Yaskawa INFORM job: DEMO_ROOF_SIDE_0625_3PAINT_10.JBI

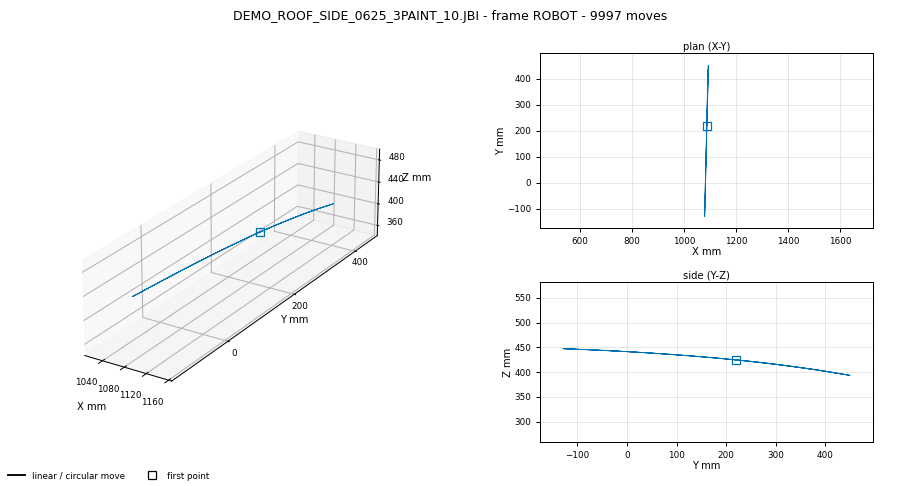
[picture p0: tool path of DEMO_ROOF_SIDE_0625_3PAINT_10.JBI in frame ROBOT, 9997 of 9997 moves have a stored position in this frame; points joined in program order, loops and branches not executed]
/JOB
//NAME DEMO_ROOF_SIDE_0625_3PAINT10
//POS
///NPOS 9997,0,0,0,0,0
///TOOL 0
///USER 0
///POSTYPE ROBOT
///RECTAN
///RCONF 1,0,0,0,0,0,0,0,0,0,0,0,0,0,0,0,0,0,0,0,0,0,0,0
C00000=1088.381,219.309,425.183,176.120,21.168,153.279
C00001=1088.386,219.557,425.158,176.123,21.170,153.279
C00002=1088.393,219.806,425.133,176.125,21.172,153.279
C00003=1088.398,220.056,425.108,176.128,21.175,153.279
C00004=1088.403,220.304,425.083,176.131,21.177,153.279
C00005=1088.409,220.553,425.058,176.134,21.180,153.280
C00006=1088.415,220.801,425.033,176.136,21.182,153.280
C00007=1088.420,221.050,425.007,176.140,21.184,153.280
C00008=1088.426,221.299,424.982,176.142,21.187,153.280
C00009=1088.432,221.547,424.957,176.145,21.189,153.280
C00010=1088.437,221.796,424.931,176.147,21.192,153.280
C00011=1088.446,222.184,424.893,176.152,21.195,153.280
C00012=1088.455,222.571,424.853,176.156,21.199,153.280
C00013=1088.463,222.958,424.814,176.160,21.203,153.280
C00014=1088.472,223.347,424.775,176.164,21.207,153.281
C00015=1088.478,223.596,424.749,176.167,21.209,153.281
C00016=1088.483,223.844,424.724,176.170,21.212,153.281
C00017=1088.490,224.092,424.698,176.173,21.214,153.281
C00018=1088.495,224.342,424.673,176.175,21.217,153.281
C00019=1088.500,224.590,424.648,176.178,21.219,153.281
C00020=1088.506,224.839,424.622,176.181,21.222,153.281
C00021=1088.511,225.087,424.597,176.184,21.224,153.281
C00022=1088.517,225.336,424.571,176.187,21.227,153.281
C00023=1088.523,225.584,424.546,176.189,21.229,153.281
C00024=1088.528,225.833,424.521,176.192,21.231,153.281
C00025=1088.534,226.082,424.496,176.195,21.233,153.281
C00026=1088.539,226.331,424.470,176.198,21.236,153.282
C00027=1088.546,226.580,424.445,176.200,21.238,153.282
C00028=1088.550,226.828,424.419,176.203,21.241,153.282
C00029=1088.557,227.077,424.394,176.205,21.243,153.282
C00030=1088.562,227.326,424.368,176.208,21.246,153.282
C00031=1088.568,227.574,424.343,176.211,21.248,153.282
C00032=1088.573,227.823,424.317,176.214,21.251,153.282
C00033=1088.579,228.071,424.292,176.217,21.253,153.282
C00034=1088.585,228.320,424.266,176.219,21.255,153.282
C00035=1088.590,228.568,424.241,176.222,21.258,153.282
C00036=1088.596,228.817,424.215,176.225,21.260,153.283
C00037=1088.601,229.066,424.189,176.228,21.263,153.283
C00038=1088.608,229.315,424.163,176.230,21.265,153.283
C00039=1088.612,229.563,424.138,176.233,21.268,153.283
C00040=1088.619,229.811,424.112,176.236,21.270,153.283
C00041=1088.624,230.060,424.086,176.239,21.273,153.283
C00042=1088.631,230.309,424.061,176.242,21.275,153.283
C00043=1088.636,230.558,424.035,176.244,21.277,153.283
C00044=1088.641,230.806,424.009,176.247,21.280,153.283
C00045=1088.646,231.055,423.983,176.250,21.282,153.283
C00046=1088.653,231.304,423.958,176.253,21.285,153.283
C00047=1088.658,231.552,423.931,176.255,21.287,153.284
C00048=1088.663,231.800,423.906,176.258,21.289,153.284
C00049=1088.669,232.049,423.880,176.261,21.292,153.284
C00050=1088.675,232.298,423.854,176.264,21.295,153.284
C00051=1088.680,232.547,423.828,176.267,21.297,153.284
C00052=1088.686,232.795,423.802,176.269,21.299,153.284
C00053=1088.692,233.043,423.777,176.272,21.302,153.284
C00054=1088.697,233.292,423.751,176.275,21.305,153.284
C00055=1088.703,233.541,423.724,176.278,21.307,153.284
C00056=1088.709,233.790,423.698,176.281,21.310,153.284
C00057=1088.714,234.039,423.672,176.283,21.312,153.285
C00058=1088.720,234.287,423.647,176.286,21.314,153.285
C00059=1088.725,234.535,423.621,176.288,21.317,153.285
C00060=1088.731,234.784,423.595,176.292,21.319,153.285
C00061=1088.737,235.032,423.568,176.295,21.322,153.285
C00062=1088.742,235.281,423.542,176.297,21.324,153.285
C00063=1088.751,235.661,423.502,176.302,21.328,153.285
C00064=1088.759,236.040,423.463,176.306,21.332,153.285
C00065=1088.768,236.419,423.422,176.310,21.336,153.286
C00066=1088.776,236.797,423.383,176.314,21.339,153.286
C00067=1088.782,237.046,423.357,176.317,21.342,153.286
C00068=1088.788,237.295,423.331,176.319,21.345,153.286
C00069=1088.793,237.544,423.305,176.323,21.347,153.286
C00070=1088.799,237.792,423.278,176.326,21.350,153.286
C00071=1088.804,238.041,423.252,176.328,21.352,153.286
C00072=1088.810,238.289,423.225,176.331,21.355,153.286
C00073=1088.816,238.538,423.199,176.334,21.357,153.286
C00074=1088.821,238.786,423.174,176.337,21.359,153.286
C00075=1088.827,239.034,423.147,176.340,21.362,153.287
C00076=1088.833,239.283,423.121,176.342,21.364,153.287
C00077=1088.838,239.531,423.094,176.345,21.367,153.287
C00078=1088.844,239.780,423.069,176.348,21.369,153.287
C00079=1088.850,240.029,423.042,176.350,21.372,153.287
C00080=1088.855,240.277,423.015,176.354,21.375,153.287
C00081=1088.861,240.526,422.989,176.357,21.377,153.287
C00082=1088.867,240.774,422.963,176.359,21.379,153.287
C00083=1088.873,241.023,422.936,176.362,21.382,153.287
C00084=1088.878,241.272,422.910,176.364,21.384,153.288
C00085=1088.884,241.520,422.883,176.368,21.387,153.288
C00086=1088.890,241.769,422.857,176.371,21.389,153.288
C00087=1088.895,242.017,422.830,176.373,21.392,153.288
C00088=1088.901,242.266,422.804,176.376,21.394,153.288
C00089=1088.906,242.515,422.777,176.379,21.397,153.288
C00090=1088.912,242.763,422.750,176.382,21.399,153.288
C00091=1088.917,243.011,422.724,176.385,21.402,153.288
C00092=1088.923,243.260,422.698,176.388,21.405,153.288
C00093=1088.929,243.509,422.671,176.390,21.407,153.288
C00094=1088.934,243.757,422.644,176.393,21.410,153.289
C00095=1088.940,244.005,422.618,176.396,21.412,153.289
C00096=1088.945,244.254,422.591,176.399,21.414,153.289
C00097=1088.951,244.502,422.564,176.402,21.417,153.289
C00098=1088.956,244.751,422.538,176.405,21.420,153.289
C00099=1088.962,245.000,422.511,176.407,21.422,153.289
C00100=1088.969,245.249,422.484,176.410,21.425,153.289
C00101=1088.974,245.497,422.457,176.413,21.428,153.289
C00102=1088.979,245.746,422.430,176.416,21.430,153.289
C00103=1088.985,245.994,422.404,176.419,21.432,153.290
C00104=1088.991,246.242,422.377,176.422,21.435,153.290
C00105=1088.996,246.491,422.350,176.424,21.437,153.290
C00106=1089.002,246.740,422.323,176.427,21.440,153.290
C00107=1089.008,246.988,422.297,176.430,21.443,153.290
C00108=1089.013,247.237,422.269,176.433,21.445,153.290
C00109=1089.018,247.485,422.243,176.436,21.448,153.290
C00110=1089.024,247.733,422.216,176.439,21.451,153.290
C00111=1089.029,247.982,422.189,176.441,21.453,153.291
C00112=1089.035,248.230,422.162,176.444,21.455,153.291
C00113=1089.040,248.479,422.135,176.447,21.458,153.291
C00114=1089.046,248.728,422.108,176.450,21.461,153.291
C00115=1089.055,249.100,422.068,176.454,21.465,153.291
C00116=1089.063,249.472,422.027,176.458,21.468,153.291
C00117=1089.071,249.844,421.987,176.463,21.473,153.291
C00118=1089.079,250.216,421.946,176.467,21.476,153.292
C00119=1089.085,250.465,421.919,176.470,21.479,153.292
C00120=1089.091,250.713,421.891,176.473,21.482,153.292
C00121=1089.096,250.962,421.865,176.476,21.484,153.292
C00122=1089.101,251.210,421.837,176.478,21.487,153.292
C00123=1089.107,251.459,421.811,176.481,21.489,153.292
C00124=1089.113,251.707,421.783,176.484,21.492,153.292
C00125=1089.118,251.955,421.756,176.487,21.495,153.293
C00126=1089.124,252.204,421.728,176.490,21.497,153.293
C00127=1089.130,252.453,421.702,176.493,21.500,153.293
C00128=1089.135,252.701,421.674,176.496,21.503,153.293
C00129=1089.141,252.949,421.647,176.498,21.505,153.293
C00130=1089.146,253.198,421.620,176.501,21.508,153.293
C00131=1089.153,253.446,421.592,176.504,21.510,153.293
C00132=1089.158,253.695,421.565,176.507,21.513,153.293
C00133=1089.163,253.944,421.538,176.510,21.515,153.294
C00134=1089.169,254.191,421.510,176.513,21.518,153.294
C00135=1089.174,254.441,421.483,176.516,21.521,153.294
C00136=1089.180,254.689,421.455,176.518,21.523,153.294
C00137=1089.185,254.937,421.428,176.521,21.526,153.294
C00138=1089.191,255.186,421.401,176.525,21.528,153.294
C00139=1089.197,255.434,421.373,176.528,21.531,153.294
C00140=1089.203,255.683,421.346,176.530,21.534,153.294
C00141=1089.208,255.931,421.319,176.533,21.536,153.295
C00142=1089.213,256.179,421.291,176.536,21.539,153.295
C00143=1089.220,256.428,421.264,176.538,21.541,153.295
C00144=1089.225,256.676,421.236,176.541,21.544,153.295
C00145=1089.231,256.924,421.209,176.545,21.547,153.295
C00146=1089.237,257.174,421.181,176.548,21.549,153.295
C00147=1089.242,257.422,421.153,176.550,21.552,153.295
C00148=1089.248,257.669,421.126,176.553,21.555,153.295
C00149=1089.254,257.919,421.098,176.556,21.557,153.296
C00150=1089.259,258.167,421.070,176.559,21.560,153.296
C00151=1089.265,258.415,421.044,176.562,21.562,153.296
C00152=1089.271,258.664,421.015,176.565,21.565,153.296
C00153=1089.277,258.912,420.988,176.568,21.567,153.296
C00154=1089.282,259.160,420.961,176.571,21.570,153.296
C00155=1089.288,259.409,420.933,176.573,21.573,153.296
C00156=1089.294,259.657,420.905,176.576,21.575,153.296
C00157=1089.299,259.905,420.878,176.580,21.578,153.296
C00158=1089.305,260.154,420.850,176.583,21.581,153.297
C00159=1089.311,260.402,420.822,176.585,21.583,153.297
C00160=1089.317,260.651,420.795,176.588,21.586,153.297
C00161=1089.322,260.899,420.767,176.591,21.588,153.297
C00162=1089.328,261.147,420.739,176.594,21.591,153.297
C00163=1089.334,261.396,420.711,176.597,21.594,153.297
C00164=1089.339,261.644,420.683,176.600,21.596,153.297
C00165=1089.345,261.893,420.655,176.603,21.599,153.297
C00166=1089.351,262.141,420.628,176.606,21.602,153.298
C00167=1089.360,262.510,420.586,176.610,21.605,153.298
C00168=1089.369,262.880,420.545,176.614,21.609,153.298
C00169=1089.377,263.249,420.503,176.619,21.614,153.298
C00170=1089.386,263.618,420.461,176.623,21.617,153.298
C00171=1089.391,263.867,420.434,176.626,21.620,153.299
C00172=1089.397,264.115,420.406,176.629,21.623,153.299
C00173=1089.403,264.364,420.378,176.632,21.625,153.299
C00174=1089.409,264.612,420.350,176.635,21.627,153.299
C00175=1089.414,264.860,420.322,176.638,21.630,153.299
C00176=1089.420,265.109,420.294,176.641,21.633,153.299
C00177=1089.425,265.357,420.266,176.644,21.636,153.299
C00178=1089.431,265.606,420.238,176.647,21.639,153.300
C00179=1089.437,265.854,420.210,176.649,21.641,153.300
C00180=1089.442,266.102,420.181,176.652,21.644,153.300
C00181=1089.448,266.350,420.153,176.655,21.646,153.300
C00182=1089.454,266.599,420.125,176.659,21.649,153.300
C00183=1089.459,266.847,420.097,176.662,21.652,153.300
C00184=1089.465,267.095,420.068,176.664,21.654,153.300
C00185=1089.471,267.343,420.040,176.667,21.657,153.301
C00186=1089.477,267.592,420.012,176.670,21.660,153.301
C00187=1089.482,267.840,419.984,176.673,21.663,153.301
C00188=1089.488,268.089,419.955,176.676,21.666,153.301
C00189=1089.493,268.337,419.928,176.678,21.668,153.301
C00190=1089.499,268.586,419.899,176.681,21.671,153.301
C00191=1089.505,268.833,419.871,176.685,21.673,153.301
C00192=1089.511,269.082,419.842,176.688,21.676,153.302
C00193=1089.516,269.330,419.814,176.691,21.679,153.302
C00194=1089.522,269.579,419.786,176.694,21.682,153.302
C00195=1089.527,269.827,419.757,176.696,21.684,153.302
C00196=1089.533,270.075,419.728,176.699,21.687,153.302
C00197=1089.538,270.323,419.700,176.702,21.690,153.302
C00198=1089.544,270.572,419.672,176.705,21.693,153.302
C00199=1089.550,270.820,419.643,176.708,21.696,153.303
C00200=1089.556,271.068,419.615,176.712,21.699,153.303
C00201=1089.561,271.317,419.586,176.714,21.701,153.303
C00202=1089.567,271.565,419.557,176.717,21.704,153.303
C00203=1089.573,271.813,419.529,176.720,21.707,153.303
C00204=1089.579,272.062,419.501,176.723,21.709,153.303
C00205=1089.584,272.310,419.472,176.726,21.712,153.304
C00206=1089.590,272.558,419.444,176.729,21.715,153.304
C00207=1089.595,272.806,419.415,176.731,21.718,153.304
C00208=1089.601,273.055,419.386,176.734,21.720,153.304
C00209=1089.607,273.304,419.358,176.737,21.723,153.304
C00210=1089.613,273.551,419.329,176.741,21.726,153.304
C00211=1089.618,273.800,419.300,176.744,21.729,153.305
C00212=1089.623,274.048,419.272,176.747,21.732,153.305
C00213=1089.629,274.296,419.243,176.750,21.735,153.305
C00214=1089.635,274.545,419.214,176.752,21.737,153.305
C00215=1089.640,274.793,419.186,176.755,21.740,153.305
C00216=1089.646,275.041,419.157,176.758,21.743,153.305
C00217=1089.652,275.289,419.127,176.761,21.745,153.306
C00218=1089.657,275.537,419.099,176.764,21.748,153.306
C00219=1089.666,275.910,419.056,176.769,21.753,153.306
C00220=1089.674,276.282,419.012,176.773,21.756,153.306
C00221=1089.683,276.654,418.969,176.777,21.761,153.307
C00222=1089.692,277.027,418.926,176.782,21.765,153.307
C00223=1089.697,277.274,418.897,176.785,21.768,153.307
C00224=1089.703,277.522,418.868,176.788,21.771,153.307
C00225=1089.709,277.771,418.839,176.791,21.773,153.307
C00226=1089.714,278.019,418.810,176.794,21.777,153.308
C00227=1089.720,278.267,418.781,176.796,21.779,153.308
C00228=1089.726,278.515,418.752,176.799,21.782,153.308
C00229=1089.731,278.764,418.723,176.802,21.785,153.308
C00230=1089.737,279.012,418.694,176.806,21.788,153.308
C00231=1089.742,279.260,418.665,176.809,21.790,153.308
C00232=1089.749,279.508,418.636,176.812,21.793,153.309
C00233=1089.754,279.756,418.606,176.815,21.796,153.309
C00234=1089.759,280.005,418.578,176.818,21.799,153.309
C00235=1089.765,280.253,418.548,176.821,21.802,153.309
C00236=1089.771,280.501,418.519,176.823,21.805,153.309
C00237=1089.776,280.749,418.490,176.826,21.808,153.310
C00238=1089.782,280.997,418.461,176.829,21.810,153.310
C00239=1089.788,281.246,418.431,176.832,21.813,153.310
C00240=1089.794,281.494,418.402,176.835,21.816,153.310
C00241=1089.800,281.742,418.373,176.838,21.819,153.310
C00242=1089.805,281.990,418.345,176.841,21.822,153.310
C00243=1089.811,282.239,418.315,176.844,21.825,153.311
C00244=1089.816,282.487,418.285,176.847,21.828,153.311
C00245=1089.822,282.735,418.256,176.851,21.831,153.311
C00246=1089.827,282.983,418.227,176.853,21.834,153.311
C00247=1089.833,283.232,418.197,176.856,21.836,153.311
C00248=1089.839,283.480,418.168,176.859,21.839,153.312
C00249=1089.844,283.728,418.139,176.862,21.842,153.312
C00250=1089.850,283.976,418.108,176.865,21.845,153.312
C00251=1089.856,284.223,418.080,176.868,21.848,153.312
C00252=1089.861,284.472,418.050,176.871,21.851,153.312
C00253=1089.867,284.720,418.021,176.874,21.854,153.313
C00254=1089.872,284.969,417.991,176.877,21.857,153.313
C00255=1089.879,285.217,417.962,176.880,21.860,153.313
C00256=1089.884,285.465,417.932,176.883,21.863,153.313
C00257=1089.890,285.714,417.903,176.886,21.866,153.313
C00258=1089.895,285.961,417.874,176.889,21.869,153.314
C00259=1089.901,286.209,417.844,176.892,21.872,153.314
C00260=1089.907,286.457,417.814,176.895,21.875,153.314
C00261=1089.912,286.706,417.784,176.898,21.877,153.314
C00262=1089.918,286.954,417.755,176.900,21.880,153.314
C00263=1089.924,287.202,417.725,176.903,21.883,153.315
C00264=1089.930,287.450,417.695,176.907,21.886,153.315
C00265=1089.935,287.699,417.666,176.910,21.889,153.315
C00266=1089.942,287.947,417.637,176.913,21.892,153.315
C00267=1089.947,288.195,417.606,176.916,21.895,153.315
C00268=1089.953,288.443,417.577,176.919,21.898,153.316
C00269=1089.958,288.691,417.547,176.922,21.901,153.316
C00270=1089.964,288.939,417.517,176.925,21.904,153.316
C00271=1089.973,289.320,417.471,176.929,21.908,153.316
C00272=1089.982,289.702,417.425,176.934,21.913,153.317
C00273=1089.991,290.083,417.380,176.938,21.917,153.317
C00274=1089.999,290.465,417.334,176.943,21.922,153.317
C00275=1090.004,290.714,417.304,176.946,21.925,153.318
C00276=1090.010,290.962,417.274,176.949,21.928,153.318
C00277=1090.017,291.210,417.245,176.952,21.931,153.318
C00278=1090.022,291.458,417.214,176.955,21.934,153.318
C00279=1090.028,291.706,417.185,176.958,21.937,153.318
C00280=1090.034,291.954,417.154,176.961,21.940,153.319
C00281=1090.039,292.202,417.125,176.964,21.943,153.319
C00282=1090.045,292.450,417.094,176.967,21.946,153.319
C00283=1090.051,292.698,417.064,176.970,21.949,153.319
C00284=1090.056,292.946,417.034,176.973,21.952,153.320
C00285=1090.062,293.194,417.004,176.976,21.955,153.320
C00286=1090.068,293.443,416.974,176.979,21.958,153.320
C00287=1090.073,293.690,416.944,176.982,21.961,153.320
C00288=1090.079,293.938,416.914,176.985,21.964,153.321
C00289=1090.085,294.187,416.884,176.988,21.968,153.321
C00290=1090.090,294.435,416.853,176.991,21.970,153.321
C00291=1090.096,294.683,416.823,176.994,21.974,153.321
C00292=1090.101,294.931,416.793,176.997,21.977,153.321
C00293=1090.107,295.179,416.763,177.000,21.980,153.322
C00294=1090.113,295.427,416.732,177.003,21.983,153.322
C00295=1090.119,295.675,416.702,177.006,21.986,153.322
C00296=1090.124,295.923,416.672,177.009,21.989,153.322
C00297=1090.131,296.172,416.642,177.012,21.992,153.323
C00298=1090.136,296.419,416.611,177.015,21.995,153.323
C00299=1090.142,296.667,416.581,177.018,21.998,153.323
C00300=1090.147,296.916,416.551,177.022,22.001,153.323
C00301=1090.153,297.164,416.520,177.025,22.005,153.324
C00302=1090.159,297.412,416.490,177.028,22.008,153.324
C00303=1090.164,297.659,416.460,177.031,22.011,153.324
C00304=1090.170,297.907,416.429,177.034,22.014,153.324
C00305=1090.176,298.155,416.399,177.037,22.017,153.325
C00306=1090.181,298.403,416.368,177.040,22.020,153.325
C00307=1090.187,298.651,416.338,177.043,22.024,153.325
C00308=1090.192,298.900,416.307,177.046,22.026,153.325
C00309=1090.198,299.148,416.277,177.049,22.030,153.326
C00310=1090.204,299.396,416.246,177.052,22.033,153.326
C00311=1090.209,299.644,416.215,177.054,22.036,153.326
C00312=1090.215,299.892,416.185,177.058,22.039,153.326
C00313=1090.220,300.140,416.154,177.060,22.042,153.327
C00314=1090.226,300.388,416.124,177.063,22.046,153.327
C00315=1090.232,300.636,416.093,177.066,22.049,153.327
C00316=1090.237,300.884,416.063,177.069,22.052,153.328
C00317=1090.243,301.131,416.031,177.072,22.055,153.328
C00318=1090.248,301.380,416.000,177.075,22.058,153.328
C00319=1090.254,301.628,415.970,177.078,22.062,153.328
C00320=1090.259,301.876,415.939,177.082,22.065,153.329
C00321=1090.265,302.124,415.908,177.085,22.068,153.329
C00322=1090.271,302.372,415.878,177.088,22.072,153.329
C00323=1090.280,302.767,415.828,177.092,22.077,153.330
C00324=1090.289,303.162,415.779,177.097,22.082,153.330
C00325=1090.298,303.559,415.730,177.102,22.087,153.331
C00326=1090.307,303.954,415.681,177.107,22.092,153.331
C00327=1090.312,304.202,415.650,177.110,22.096,153.331
C00328=1090.319,304.450,415.619,177.113,22.099,153.332
C00329=1090.324,304.698,415.588,177.116,22.102,153.332
C00330=1090.330,304.946,415.558,177.119,22.105,153.332
C00331=1090.335,305.193,415.526,177.122,22.108,153.332
C00332=1090.341,305.442,415.495,177.125,22.111,153.333
C00333=1090.347,305.690,415.464,177.128,22.115,153.333
C00334=1090.352,305.938,415.433,177.131,22.119,153.333
C00335=1090.358,306.185,415.402,177.134,22.122,153.334
C00336=1090.364,306.434,415.371,177.137,22.125,153.334
C00337=1090.370,306.681,415.340,177.140,22.128,153.334
C00338=1090.375,306.930,415.309,177.143,22.131,153.334
C00339=1090.381,307.178,415.278,177.146,22.134,153.335
C00340=1090.387,307.426,415.247,177.149,22.138,153.335
C00341=1090.392,307.673,415.216,177.152,22.141,153.335
C00342=1090.398,307.922,415.184,177.156,22.145,153.336
C00343=1090.403,308.170,415.153,177.159,22.148,153.336
C00344=1090.410,308.417,415.122,177.162,22.151,153.336
C00345=1090.415,308.666,415.091,177.165,22.155,153.337
C00346=1090.421,308.913,415.060,177.168,22.158,153.337
C00347=1090.427,309.161,415.028,177.170,22.161,153.337
C00348=1090.432,309.409,414.997,177.174,22.164,153.337
C00349=1090.439,309.657,414.966,177.176,22.167,153.338
C00350=1090.444,309.905,414.935,177.180,22.171,153.338
C00351=1090.450,310.153,414.903,177.183,22.174,153.338
C00352=1090.456,310.400,414.872,177.186,22.178,153.339
C00353=1090.461,310.649,414.840,177.189,22.181,153.339
C00354=1090.468,310.896,414.809,177.192,22.184,153.339
C00355=1090.473,311.145,414.778,177.195,22.187,153.340
C00356=1090.479,311.393,414.746,177.198,22.191,153.340
C00357=1090.485,311.640,414.715,177.201,22.194,153.340
C00358=1090.491,311.888,414.683,177.204,22.198,153.340
C00359=1090.496,312.137,414.652,177.207,22.201,153.341
C00360=1090.502,312.384,414.620,177.210,22.204,153.341
C00361=1090.509,312.632,414.589,177.213,22.208,153.341
C00362=1090.514,312.880,414.557,177.216,22.211,153.342
C00363=1090.520,313.129,414.526,177.219,22.214,153.342
C00364=1090.526,313.376,414.495,177.223,22.218,153.342
C00365=1090.532,313.624,414.463,177.226,22.221,153.343
C00366=1090.537,313.871,414.431,177.229,22.224,153.343
C00367=1090.543,314.120,414.399,177.232,22.228,153.343
C00368=1090.549,314.367,414.369,177.235,22.231,153.344
C00369=1090.555,314.616,414.337,177.238,22.234,153.344
C00370=1090.561,314.864,414.305,177.241,22.238,153.344
C00371=1090.566,315.111,414.273,177.244,22.241,153.344
C00372=1090.572,315.360,414.241,177.247,22.245,153.345
C00373=1090.578,315.607,414.209,177.250,22.248,153.345
C00374=1090.584,315.855,414.177,177.253,22.252,153.345
C00375=1090.592,316.253,414.127,177.258,22.258,153.346
C00376=1090.602,316.652,414.075,177.263,22.263,153.347
C00377=1090.610,317.051,414.024,177.267,22.269,153.347
C00378=1090.619,317.448,413.973,177.272,22.274,153.348
C00379=1090.625,317.696,413.941,177.275,22.278,153.348
C00380=1090.631,317.944,413.909,177.279,22.282,153.349
C00381=1090.636,318.192,413.877,177.282,22.286,153.349
C00382=1090.641,318.440,413.845,177.284,22.289,153.349
C00383=1090.647,318.688,413.813,177.287,22.293,153.350
C00384=1090.653,318.936,413.781,177.290,22.296,153.350
C00385=1090.659,319.183,413.748,177.294,22.300,153.350
C00386=1090.665,319.431,413.716,177.297,22.303,153.351
C00387=1090.670,319.679,413.685,177.300,22.307,153.351
C00388=1090.676,319.927,413.652,177.302,22.310,153.352
C00389=1090.681,320.175,413.621,177.305,22.314,153.352
C00390=1090.687,320.423,413.588,177.309,22.318,153.352
C00391=1090.693,320.671,413.556,177.312,22.321,153.353
C00392=1090.699,320.918,413.524,177.315,22.325,153.353
C00393=1090.704,321.167,413.491,177.317,22.328,153.353
C00394=1090.710,321.415,413.459,177.321,22.332,153.354
C00395=1090.716,321.662,413.427,177.324,22.336,153.354
C00396=1090.722,321.910,413.395,177.327,22.339,153.355
C00397=1090.728,322.158,413.363,177.330,22.343,153.355
C00398=1090.733,322.405,413.330,177.332,22.346,153.355
C00399=1090.739,322.654,413.298,177.336,22.350,153.356
C00400=1090.745,322.902,413.266,177.339,22.354,153.356
C00401=1090.750,323.149,413.234,177.342,22.357,153.357
C00402=1090.756,323.397,413.201,177.345,22.361,153.357
C00403=1090.762,323.645,413.168,177.348,22.365,153.357
C00404=1090.768,323.893,413.136,177.351,22.369,153.358
C00405=1090.773,324.140,413.103,177.354,22.372,153.358
C00406=1090.779,324.388,413.071,177.357,22.376,153.359
C00407=1090.785,324.637,413.039,177.360,22.380,153.359
C00408=1090.791,324.884,413.006,177.363,22.383,153.359
C00409=1090.796,325.132,412.974,177.366,22.387,153.360
C00410=1090.802,325.380,412.941,177.370,22.391,153.360
C00411=1090.808,325.627,412.909,177.373,22.394,153.360
C00412=1090.814,325.876,412.876,177.375,22.398,153.361
C00413=1090.819,326.123,412.844,177.378,22.402,153.361
C00414=1090.825,326.371,412.812,177.382,22.405,153.362
C00415=1090.831,326.619,412.778,177.385,22.409,153.362
C00416=1090.837,326.867,412.746,177.387,22.413,153.363
C00417=1090.843,327.115,412.714,177.390,22.416,153.363
C00418=1090.849,327.363,412.680,177.394,22.420,153.363
C00419=1090.854,327.610,412.649,177.397,22.424,153.364
C00420=1090.860,327.858,412.616,177.400,22.428,153.364
C00421=1090.866,328.106,412.582,177.403,22.432,153.365
C00422=1090.872,328.353,412.550,177.406,22.435,153.365
C00423=1090.877,328.602,412.517,177.409,22.439,153.365
C00424=1090.884,328.849,412.484,177.412,22.443,153.366
C00425=1090.890,329.097,412.452,177.415,22.446,153.366
C00426=1090.896,329.345,412.418,177.418,22.450,153.367
C00427=1090.905,329.736,412.367,177.423,22.456,153.367
C00428=1090.914,330.128,412.315,177.428,22.462,153.368
C00429=1090.924,330.518,412.263,177.433,22.468,153.369
C00430=1090.932,330.910,412.212,177.437,22.474,153.369
C00431=1090.939,331.158,412.179,177.441,22.478,153.370
C00432=1090.944,331.406,412.145,177.444,22.482,153.370
C00433=1090.950,331.653,412.113,177.447,22.485,153.371
C00434=1090.956,331.901,412.079,177.450,22.490,153.371
C00435=1090.962,332.149,412.047,177.453,22.493,153.371
C00436=1090.968,332.397,412.013,177.457,22.497,153.372
C00437=1090.973,332.644,411.980,177.459,22.501,153.372
C00438=1090.979,332.892,411.947,177.462,22.505,153.373
C00439=1090.985,333.140,411.914,177.466,22.509,153.373
C00440=1090.991,333.388,411.881,177.468,22.513,153.374
C00441=1090.996,333.636,411.847,177.471,22.517,153.374
C00442=1091.003,333.883,411.814,177.475,22.521,153.375
C00443=1091.008,334.131,411.781,177.477,22.525,153.375
C00444=1091.014,334.379,411.748,177.480,22.529,153.376
C00445=1091.019,334.627,411.714,177.484,22.533,153.376
C00446=1091.025,334.874,411.682,177.486,22.537,153.377
C00447=1091.031,335.122,411.649,177.490,22.541,153.377
C00448=1091.036,335.370,411.615,177.493,22.545,153.378
C00449=1091.042,335.617,411.581,177.496,22.549,153.378
C00450=1091.048,335.865,411.549,177.499,22.553,153.379
C00451=1091.054,336.113,411.515,177.502,22.557,153.379
C00452=1091.060,336.361,411.482,177.505,22.561,153.379
C00453=1091.066,336.608,411.448,177.508,22.565,153.380
C00454=1091.072,336.856,411.415,177.511,22.569,153.381
C00455=1091.078,337.104,411.381,177.514,22.573,153.381
C00456=1091.083,337.352,411.348,177.517,22.577,153.381
C00457=1091.089,337.599,411.314,177.520,22.581,153.382
C00458=1091.095,337.847,411.281,177.523,22.585,153.382
C00459=1091.100,338.095,411.247,177.526,22.589,153.383
C00460=1091.107,338.342,411.214,177.530,22.593,153.383
C00461=1091.112,338.590,411.181,177.532,22.597,153.384
C00462=1091.118,338.838,411.147,177.536,22.602,153.384
C00463=1091.124,339.085,411.113,177.539,22.606,153.385
C00464=1091.129,339.333,411.080,177.541,22.610,153.386
C00465=1091.135,339.580,411.046,177.545,22.614,153.386
C00466=1091.141,339.828,411.012,177.548,22.618,153.387
C00467=1091.147,340.076,410.978,177.551,22.622,153.387
C00468=1091.153,340.324,410.945,177.554,22.626,153.388
C00469=1091.159,340.571,410.911,177.557,22.631,153.388
C00470=1091.164,340.819,410.877,177.560,22.635,153.389
C00471=1091.170,341.066,410.843,177.564,22.639,153.389
C00472=1091.176,341.314,410.810,177.566,22.643,153.390
C00473=1091.181,341.562,410.776,177.569,22.647,153.390
C00474=1091.187,341.810,410.743,177.572,22.652,153.391
C00475=1091.194,342.058,410.708,177.575,22.655,153.391
C00476=1091.199,342.305,410.674,177.579,22.660,153.392
C00477=1091.205,342.553,410.641,177.581,22.664,153.392
C00478=1091.211,342.800,410.607,177.585,22.668,153.393
C00479=1091.219,343.186,410.554,177.590,22.675,153.394
C00480=1091.228,343.571,410.501,177.594,22.682,153.395
C00481=1091.238,343.957,410.448,177.599,22.688,153.395
C00482=1091.247,344.342,410.395,177.604,22.695,153.396
C00483=1091.253,344.590,410.362,177.607,22.699,153.397
C00484=1091.259,344.837,410.328,177.610,22.703,153.397
C00485=1091.264,345.086,410.293,177.613,22.708,153.398
C00486=1091.270,345.333,410.258,177.616,22.712,153.399
C00487=1091.276,345.580,410.224,177.619,22.716,153.399
C00488=1091.282,345.827,410.190,177.622,22.721,153.400
C00489=1091.287,346.076,410.156,177.625,22.725,153.400
C00490=1091.293,346.324,410.122,177.628,22.730,153.401
C00491=1091.299,346.571,410.088,177.631,22.734,153.401
C00492=1091.305,346.818,410.054,177.635,22.739,153.402
C00493=1091.311,347.067,410.019,177.637,22.743,153.403
C00494=1091.316,347.314,409.985,177.641,22.747,153.403
C00495=1091.322,347.561,409.951,177.643,22.751,153.404
C00496=1091.328,347.808,409.917,177.647,22.756,153.404
C00497=1091.334,348.057,409.882,177.649,22.761,153.405
C00498=1091.340,348.304,409.848,177.653,22.765,153.406
C00499=1091.346,348.551,409.814,177.655,22.769,153.406
C00500=1091.351,348.799,409.779,177.659,22.774,153.407
C00501=1091.357,349.047,409.745,177.662,22.779,153.407
C00502=1091.363,349.294,409.711,177.665,22.783,153.408
C00503=1091.368,349.542,409.676,177.668,22.788,153.409
C00504=1091.375,349.790,409.641,177.671,22.792,153.409
C00505=1091.380,350.037,409.606,177.674,22.797,153.410
C00506=1091.386,350.284,409.572,177.677,22.801,153.410
C00507=1091.392,350.532,409.538,177.680,22.806,153.411
C00508=1091.397,350.780,409.503,177.683,22.810,153.412
C00509=1091.403,351.027,409.469,177.686,22.815,153.412
C00510=1091.409,351.274,409.433,177.690,22.820,153.413
C00511=1091.415,351.522,409.399,177.692,22.824,153.414
C00512=1091.421,351.770,409.364,177.696,22.828,153.414
C00513=1091.427,352.017,409.330,177.698,22.833,153.415
C00514=1091.433,352.264,409.295,177.702,22.838,153.416
C00515=1091.439,352.512,409.260,177.705,22.842,153.416
C00516=1091.445,352.760,409.226,177.708,22.847,153.417
C00517=1091.451,353.007,409.190,177.711,22.851,153.417
C00518=1091.456,353.255,409.156,177.714,22.856,153.418
C00519=1091.462,353.502,409.122,177.717,22.861,153.419
C00520=1091.468,353.750,409.087,177.720,22.866,153.419
C00521=1091.473,353.997,409.052,177.723,22.870,153.420
C00522=1091.480,354.245,409.016,177.726,22.875,153.421
C00523=1091.485,354.492,408.982,177.729,22.879,153.421
C00524=1091.491,354.739,408.947,177.732,22.884,153.422
C00525=1091.497,354.987,408.912,177.736,22.889,153.423
C00526=1091.503,355.234,408.877,177.738,22.894,153.423
C00527=1091.508,355.482,408.842,177.742,22.898,153.424
C00528=1091.515,355.729,408.807,177.745,22.903,153.425
C00529=1091.520,355.977,408.772,177.747,22.908,153.425
C00530=1091.526,356.224,408.737,177.751,22.913,153.426
C00531=1091.535,356.613,408.683,177.755,22.920,153.427
C00532=1091.544,357.001,408.627,177.760,22.928,153.428
C00533=1091.554,357.389,408.572,177.765,22.935,153.429
C00534=1091.562,357.777,408.517,177.770,22.943,153.430
C00535=1091.569,358.024,408.482,177.773,22.948,153.431
C00536=1091.575,358.272,408.447,177.776,22.952,153.432
C00537=1091.580,358.519,408.411,177.779,22.957,153.433
C00538=1091.586,358.767,408.376,177.782,22.962,153.433
C00539=1091.593,359.014,408.341,177.785,22.967,153.434
C00540=1091.598,359.261,408.306,177.788,22.972,153.435
C00541=1091.604,359.509,408.270,177.791,22.977,153.435
C00542=1091.609,359.757,408.235,177.794,22.982,153.436
C00543=1091.616,360.004,408.200,177.797,22.987,153.437
C00544=1091.621,360.251,408.165,177.800,22.992,153.438
C00545=1091.627,360.499,408.129,177.803,22.996,153.438
C00546=1091.633,360.746,408.093,177.806,23.001,153.439
C00547=1091.639,360.993,408.058,177.810,23.006,153.440
C00548=1091.645,361.241,408.022,177.813,23.012,153.441
C00549=1091.650,361.488,407.987,177.815,23.017,153.441
C00550=1091.657,361.735,407.952,177.819,23.022,153.442
C00551=1091.662,361.982,407.916,177.822,23.027,153.443
C00552=1091.669,362.230,407.881,177.824,23.032,153.444
C00553=1091.675,362.478,407.845,177.828,23.037,153.444
C00554=1091.680,362.724,407.810,177.831,23.042,153.445
C00555=1091.686,362.972,407.774,177.834,23.047,153.446
C00556=1091.692,363.220,407.738,177.837,23.052,153.447
C00557=1091.697,363.467,407.703,177.840,23.057,153.447
C00558=1091.703,363.714,407.667,177.843,23.062,153.448
C00559=1091.710,363.962,407.631,177.846,23.067,153.449
C00560=1091.715,364.209,407.596,177.849,23.072,153.450
C00561=1091.721,364.456,407.560,177.852,23.077,153.451
C00562=1091.727,364.704,407.524,177.855,23.083,153.451
C00563=1091.733,364.951,407.488,177.858,23.087,153.452
C00564=1091.739,365.199,407.453,177.861,23.093,153.453
C00565=1091.745,365.446,407.417,177.864,23.098,153.454
C00566=1091.751,365.693,407.381,177.867,23.103,153.455
C00567=1091.757,365.940,407.345,177.871,23.109,153.455
C00568=1091.763,366.188,407.309,177.873,23.113,153.456
C00569=1091.768,366.434,407.273,177.876,23.119,153.457
C00570=1091.774,366.682,407.238,177.880,23.124,153.458
C00571=1091.780,366.930,407.201,177.883,23.130,153.459
C00572=1091.785,367.176,407.165,177.885,23.135,153.460
C00573=1091.791,367.424,407.130,177.888,23.140,153.460
C00574=1091.797,367.672,407.094,177.891,23.146,153.461
C00575=1091.804,367.919,407.057,177.895,23.151,153.462
C00576=1091.808,368.166,407.021,177.898,23.156,153.463
C00577=1091.815,368.413,406.985,177.900,23.161,153.464
C00578=1091.821,368.661,406.949,177.903,23.167,153.464
C00579=1091.827,368.908,406.913,177.907,23.172,153.465
C00580=1091.833,369.155,406.877,177.910,23.178,153.466
C00581=1091.838,369.402,406.840,177.913,23.183,153.467
C00582=1091.844,369.650,406.805,177.915,23.188,153.468
C00583=1091.854,370.053,406.746,177.920,23.197,153.469
C00584=1091.863,370.457,406.687,177.925,23.206,153.471
C00585=1091.873,370.860,406.628,177.930,23.215,153.472
C00586=1091.883,371.263,406.568,177.935,23.224,153.474
C00587=1091.889,371.511,406.532,177.939,23.230,153.474
C00588=1091.895,371.758,406.496,177.942,23.236,153.475
C00589=1091.900,372.005,406.458,177.945,23.241,153.476
C00590=1091.907,372.253,406.423,177.947,23.246,153.477
C00591=1091.913,372.500,406.386,177.950,23.252,153.478
C00592=1091.918,372.747,406.349,177.953,23.257,153.479
C00593=1091.924,372.993,406.313,177.957,23.263,153.480
C00594=1091.931,373.241,406.277,177.960,23.269,153.481
C00595=1091.936,373.489,406.240,177.963,23.274,153.482
C00596=1091.942,373.736,406.204,177.966,23.280,153.483
C00597=1091.948,373.983,406.168,177.968,23.285,153.484
C00598=1091.954,374.230,406.130,177.971,23.291,153.484
C00599=1091.960,374.477,406.094,177.975,23.297,153.485
C00600=1091.966,374.724,406.057,177.978,23.302,153.486
C00601=1091.972,374.971,406.021,177.981,23.308,153.487
C00602=1091.978,375.219,405.984,177.984,23.314,153.488
C00603=1091.984,375.465,405.947,177.987,23.320,153.489
C00604=1091.989,375.713,405.910,177.990,23.326,153.490
C00605=1091.995,375.960,405.873,177.993,23.331,153.491
C00606=1092.001,376.207,405.837,177.996,23.337,153.492
C00607=1092.007,376.454,405.800,177.998,23.342,153.493
C00608=1092.013,376.701,405.763,178.001,23.348,153.494
C00609=1092.019,376.949,405.726,178.004,23.354,153.495
C00610=1092.024,377.196,405.689,178.008,23.360,153.496
C00611=1092.031,377.443,405.653,178.011,23.366,153.497
C00612=1092.036,377.691,405.616,178.014,23.372,153.498
C00613=1092.043,377.937,405.579,178.017,23.378,153.499
C00614=1092.049,378.184,405.542,178.020,23.384,153.500
C00615=1092.054,378.432,405.505,178.023,23.390,153.501
C00616=1092.060,378.679,405.468,178.026,23.396,153.502
C00617=1092.066,378.926,405.431,178.029,23.402,153.503
C00618=1092.072,379.173,405.393,178.032,23.408,153.504
C00619=1092.078,379.420,405.357,178.035,23.414,153.505
C00620=1092.084,379.667,405.320,178.038,23.419,153.506
C00621=1092.090,379.914,405.282,178.041,23.426,153.507
C00622=1092.096,380.161,405.246,178.044,23.432,153.508
C00623=1092.102,380.408,405.209,178.047,23.438,153.509
C00624=1092.108,380.655,405.171,178.050,23.443,153.510
C00625=1092.114,380.902,405.134,178.053,23.450,153.511
C00626=1092.120,381.150,405.097,178.056,23.456,153.512
C00627=1092.125,381.396,405.060,178.059,23.462,153.513
C00628=1092.132,381.643,405.023,178.062,23.468,153.514
C00629=1092.138,381.891,404.985,178.065,23.474,153.515
C00630=1092.144,382.138,404.948,178.068,23.480,153.516
C00631=1092.150,382.385,404.910,178.071,23.486,153.517
C00632=1092.156,382.632,404.874,178.074,23.492,153.518
C00633=1092.162,382.879,404.836,178.077,23.499,153.519
C00634=1092.168,383.126,404.799,178.080,23.505,153.521
C00635=1092.173,383.342,404.766,178.082,23.510,153.521
C00636=1092.178,383.557,404.734,178.085,23.516,153.522
C00637=1092.183,383.772,404.701,178.088,23.521,153.523
C00638=1092.188,383.988,404.667,178.090,23.526,153.524
C00639=1092.193,384.203,404.635,178.093,23.532,153.525
C00640=1092.199,384.419,404.603,178.095,23.538,153.526
C00641=1092.204,384.634,404.570,178.098,23.543,153.527
C00642=1092.209,384.850,404.536,178.101,23.549,153.528
C00643=1092.215,385.097,404.499,178.103,23.555,153.529
C00644=1092.220,385.344,404.462,178.106,23.562,153.531
C00645=1092.226,385.591,404.424,178.109,23.568,153.532
C00646=1092.233,385.838,404.386,178.112,23.574,153.533
C00647=1092.238,386.086,404.349,178.116,23.581,153.534
C00648=1092.244,386.332,404.311,178.119,23.587,153.535
C00649=1092.250,386.579,404.273,178.122,23.594,153.536
C00650=1092.256,386.826,404.235,178.125,23.600,153.537
C00651=1092.263,387.073,404.197,178.128,23.607,153.538
C00652=1092.269,387.320,404.160,178.131,23.613,153.540
C00653=1092.275,387.567,404.122,178.133,23.620,153.541
C00654=1092.280,387.813,404.084,178.136,23.626,153.542
C00655=1092.286,388.060,404.046,178.139,23.633,153.543
C00656=1092.293,388.308,404.008,178.143,23.640,153.544
C00657=1092.299,388.554,403.970,178.146,23.646,153.545
C00658=1092.305,388.801,403.933,178.149,23.653,153.547
C00659=1092.311,389.049,403.894,178.152,23.659,153.548
C00660=1092.317,389.295,403.857,178.154,23.666,153.549
C00661=1092.323,389.542,403.819,178.157,23.672,153.550
C00662=1092.328,389.789,403.781,178.161,23.679,153.551
C00663=1092.335,390.037,403.743,178.164,23.686,153.553
C00664=1092.341,390.283,403.705,178.167,23.692,153.554
C00665=1092.346,390.530,403.667,178.169,23.699,153.555
C00666=1092.353,390.777,403.629,178.172,23.706,153.556
C00667=1092.359,391.024,403.590,178.175,23.713,153.558
C00668=1092.366,391.271,403.552,178.179,23.720,153.559
C00669=1092.372,391.518,403.515,178.182,23.726,153.560
C00670=1092.377,391.765,403.476,178.185,23.733,153.561
C00671=1092.383,392.012,403.438,178.187,23.740,153.562
C00672=1092.389,392.258,403.400,178.190,23.746,153.564
C00673=1092.396,392.506,403.361,178.193,23.753,153.565
C00674=1092.401,392.753,403.323,178.196,23.761,153.566
C00675=1092.407,392.999,403.285,178.199,23.767,153.567
C00676=1092.414,393.246,403.247,178.202,23.774,153.569
C00677=1092.419,393.494,403.208,178.205,23.781,153.570
C00678=1092.426,393.740,403.169,178.208,23.789,153.571
C00679=1092.432,393.987,403.132,178.211,23.795,153.573
C00680=1092.437,394.234,403.093,178.214,23.802,153.574
C00681=1092.444,394.481,403.054,178.217,23.809,153.575
C00682=1092.449,394.727,403.015,178.220,23.816,153.576
C00683=1092.456,394.975,402.977,178.223,23.824,153.578
C00684=1092.462,395.221,402.939,178.226,23.830,153.579
C00685=1092.468,395.469,402.900,178.229,23.838,153.580
C00686=1092.474,395.715,402.862,178.231,23.845,153.582
C00687=1092.480,395.963,402.823,178.235,23.852,153.583
C00688=1092.486,396.209,402.784,178.238,23.859,153.584
C00689=1092.492,396.457,402.746,178.240,23.866,153.586
C00690=1092.498,396.703,402.707,178.244,23.874,153.587
C00691=1092.503,396.925,402.672,178.246,23.880,153.589
C00692=1092.508,397.146,402.637,178.249,23.886,153.590
C00693=1092.514,397.369,402.602,178.252,23.893,153.591
C00694=1092.519,397.592,402.567,178.254,23.900,153.592
C00695=1092.525,397.814,402.532,178.256,23.906,153.593
C00696=1092.530,398.035,402.497,178.259,23.913,153.595
C00697=1092.536,398.257,402.463,178.262,23.920,153.596
C00698=1092.541,398.480,402.428,178.265,23.926,153.597
C00699=1092.547,398.727,402.389,178.268,23.933,153.599
C00700=1092.553,398.973,402.350,178.270,23.941,153.600
C00701=1092.560,399.220,402.311,178.274,23.949,153.601
C00702=1092.566,399.467,402.271,178.276,23.956,153.603
C00703=1092.572,399.714,402.234,178.279,23.963,153.604
C00704=1092.578,399.961,402.194,178.283,23.971,153.606
C00705=1092.584,400.208,402.155,178.285,23.978,153.607
C00706=1092.589,400.454,402.116,178.288,23.986,153.609
C00707=1092.596,400.701,402.077,178.291,23.993,153.610
C00708=1092.601,400.948,402.038,178.294,24.001,153.611
C00709=1092.608,401.195,401.998,178.297,24.009,153.613
C00710=1092.614,401.442,401.959,178.300,24.016,153.614
C00711=1092.620,401.688,401.920,178.303,24.024,153.616
C00712=1092.626,401.935,401.881,178.306,24.032,153.617
C00713=1092.632,402.182,401.842,178.309,24.040,153.619
C00714=1092.638,402.430,401.802,178.312,24.048,153.620
C00715=1092.643,402.676,401.763,178.315,24.055,153.622
C00716=1092.650,402.923,401.724,178.318,24.063,153.623
C00717=1092.657,403.169,401.684,178.321,24.071,153.625
C00718=1092.663,403.416,401.645,178.323,24.078,153.626
C00719=1092.668,403.663,401.606,178.327,24.086,153.628
C00720=1092.674,403.910,401.566,178.329,24.094,153.629
C00721=1092.681,404.157,401.527,178.333,24.102,153.631
C00722=1092.687,404.403,401.487,178.335,24.110,153.632
C00723=1092.694,404.651,401.448,178.339,24.118,153.634
C00724=1092.699,404.897,401.409,178.341,24.126,153.636
C00725=1092.705,405.143,401.369,178.345,24.134,153.637
C00726=1092.711,405.391,401.329,178.347,24.142,153.639
C00727=1092.718,405.638,401.290,178.350,24.150,153.640
C00728=1092.724,405.884,401.249,178.353,24.158,153.642
C00729=1092.729,406.131,401.210,178.356,24.166,153.643
C00730=1092.735,406.378,401.171,178.359,24.174,153.645
C00731=1092.742,406.624,401.131,178.362,24.182,153.647
C00732=1092.748,406.871,401.091,178.365,24.190,153.648
C00733=1092.754,407.118,401.051,178.368,24.199,153.650
C00734=1092.760,407.365,401.012,178.371,24.207,153.652
C00735=1092.766,407.611,400.972,178.374,24.215,153.653
C00736=1092.772,407.858,400.932,178.377,24.224,153.655
C00737=1092.778,408.105,400.892,178.379,24.232,153.656
C00738=1092.784,408.351,400.852,178.383,24.240,153.658
C00739=1092.790,408.599,400.812,178.385,24.248,153.660
C00740=1092.797,408.845,400.772,178.389,24.257,153.661
C00741=1092.803,409.092,400.733,178.392,24.266,153.663
C00742=1092.808,409.339,400.692,178.394,24.274,153.665
C00743=1092.815,409.586,400.652,178.398,24.283,153.667
C00744=1092.821,409.831,400.612,178.401,24.291,153.668
C00745=1092.827,410.078,400.573,178.403,24.300,153.670
C00746=1092.832,410.325,400.532,178.407,24.308,153.672
C00747=1092.838,410.548,400.496,178.409,24.316,153.673
C00748=1092.844,410.770,400.460,178.412,24.324,153.675
C00749=1092.849,410.993,400.423,178.414,24.331,153.676
C00750=1092.855,411.215,400.387,178.417,24.339,153.678
C00751=1092.860,411.438,400.351,178.419,24.347,153.679
C00752=1092.866,411.660,400.315,178.423,24.355,153.681
C00753=1092.871,411.883,400.278,178.425,24.363,153.683
C00754=1092.877,412.105,400.242,178.428,24.371,153.684
C00755=1092.883,412.352,400.202,178.431,24.380,153.686
C00756=1092.889,412.599,400.162,178.433,24.388,153.688
C00757=1092.896,412.845,400.121,178.437,24.397,153.689
C00758=1092.901,413.092,400.081,178.440,24.406,153.691
C00759=1092.908,413.338,400.040,178.443,24.415,153.693
C00760=1092.914,413.585,400.000,178.446,24.423,153.695
C00761=1092.920,413.831,399.959,178.449,24.432,153.697
C00762=1092.927,414.078,399.918,178.452,24.441,153.698
C00763=1092.933,414.325,399.878,178.455,24.450,153.700
C00764=1092.939,414.572,399.837,178.458,24.459,153.702
C00765=1092.945,414.818,399.797,178.461,24.468,153.704
C00766=1092.952,415.065,399.757,178.464,24.477,153.706
C00767=1092.958,415.311,399.716,178.467,24.487,153.708
C00768=1092.964,415.558,399.676,178.470,24.495,153.709
C00769=1092.970,415.805,399.634,178.473,24.505,153.711
C00770=1092.977,416.052,399.594,178.475,24.514,153.713
C00771=1092.983,416.298,399.553,178.479,24.523,153.715
C00772=1092.989,416.544,399.513,178.482,24.532,153.717
C00773=1092.995,416.791,399.472,178.485,24.541,153.719
C00774=1093.001,417.037,399.431,178.488,24.551,153.721
C00775=1093.007,417.284,399.390,178.491,24.560,153.723
C00776=1093.014,417.531,399.349,178.494,24.570,153.725
C00777=1093.020,417.777,399.308,178.497,24.579,153.726
C00778=1093.026,418.023,399.267,178.499,24.588,153.729
C00779=1093.032,418.270,399.227,178.503,24.598,153.730
C00780=1093.038,418.516,399.185,178.506,24.607,153.732
C00781=1093.044,418.764,399.144,178.509,24.617,153.734
C00782=1093.051,419.010,399.103,178.512,24.626,153.736
C00783=1093.057,419.256,399.063,178.515,24.636,153.738
C00784=1093.063,419.503,399.021,178.518,24.645,153.740
C00785=1093.070,419.749,398.980,178.521,24.655,153.742
C00786=1093.076,419.996,398.939,178.524,24.665,153.744
C00787=1093.082,420.242,398.898,178.527,24.675,153.746
C00788=1093.088,420.488,398.856,178.530,24.684,153.748
C00789=1093.095,420.735,398.815,178.533,24.694,153.750
C00790=1093.101,420.982,398.774,178.536,24.704,153.752
C00791=1093.106,421.228,398.733,178.539,24.714,153.755
C00792=1093.113,421.475,398.691,178.542,24.724,153.757
C00793=1093.120,421.721,398.650,178.545,24.733,153.759
C00794=1093.126,421.967,398.609,178.548,24.744,153.761
C00795=1093.132,422.214,398.567,178.551,24.753,153.763
C00796=1093.138,422.461,398.526,178.554,24.763,153.765
C00797=1093.145,422.707,398.485,178.557,24.773,153.767
C00798=1093.151,422.954,398.443,178.560,24.783,153.769
C00799=1093.157,423.200,398.402,178.563,24.793,153.771
C00800=1093.164,423.447,398.360,178.567,24.804,153.773
C00801=1093.170,423.693,398.319,178.570,24.814,153.775
C00802=1093.176,423.938,398.277,178.573,24.824,153.778
C00803=1093.182,424.169,398.238,178.575,24.834,153.780
C00804=1093.187,424.399,398.199,178.578,24.843,153.782
C00805=1093.193,424.628,398.160,178.581,24.853,153.784
C00806=1093.198,424.858,398.121,178.584,24.863,153.786
C00807=1093.205,425.088,398.082,178.586,24.872,153.788
C00808=1093.211,425.318,398.044,178.589,24.882,153.790
C00809=1093.216,425.547,398.004,178.592,24.892,153.792
C00810=1093.223,425.777,397.965,178.595,24.902,153.794
C00811=1093.229,426.024,397.924,178.598,24.912,153.796
C00812=1093.235,426.270,397.881,178.601,24.922,153.798
C00813=1093.241,426.516,397.840,178.604,24.933,153.801
C00814=1093.248,426.763,397.798,178.607,24.944,153.803
C00815=1093.254,427.009,397.756,178.611,24.955,153.805
C00816=1093.260,427.256,397.714,178.614,24.965,153.808
C00817=1093.266,427.501,397.671,178.616,24.976,153.810
C00818=1093.273,427.748,397.630,178.619,24.986,153.812
C00819=1093.279,427.994,397.587,178.622,24.997,153.814
C00820=1093.286,428.241,397.546,178.626,25.008,153.817
C00821=1093.292,428.486,397.503,178.629,25.019,153.819
C00822=1093.298,428.733,397.462,178.631,25.029,153.821
C00823=1093.305,428.980,397.419,178.634,25.040,153.824
C00824=1093.312,429.225,397.377,178.638,25.052,153.826
C00825=1093.317,429.472,397.335,178.641,25.063,153.828
C00826=1093.324,429.718,397.292,178.644,25.073,153.831
C00827=1093.330,429.964,397.250,178.647,25.085,153.833
C00828=1093.336,430.211,397.208,178.650,25.096,153.836
C00829=1093.343,430.457,397.165,178.653,25.107,153.838
C00830=1093.349,430.703,397.123,178.656,25.119,153.840
C00831=1093.356,430.949,397.080,178.659,25.129,153.843
C00832=1093.361,431.196,397.038,178.662,25.140,153.845
C00833=1093.368,431.442,396.996,178.665,25.152,153.848
C00834=1093.375,431.688,396.953,178.668,25.163,153.850
C00835=1093.381,431.935,396.910,178.671,25.175,153.853
C00836=1093.387,432.180,396.868,178.674,25.187,153.855
C00837=1093.394,432.426,396.826,178.677,25.197,153.858
C00838=1093.400,432.673,396.782,178.681,25.209,153.860
C00839=1093.407,432.919,396.740,178.683,25.221,153.863
C00840=1093.413,433.165,396.698,178.686,25.232,153.865
C00841=1093.419,433.412,396.655,178.690,25.244,153.868
C00842=1093.425,433.658,396.611,178.692,25.256,153.870
C00843=1093.432,433.904,396.569,178.696,25.268,153.873
C00844=1093.438,434.150,396.525,178.698,25.279,153.876
C00845=1093.445,434.396,396.483,178.702,25.291,153.878
C00846=1093.450,434.642,396.440,178.705,25.303,153.881
C00847=1093.457,434.888,396.398,178.708,25.315,153.883
C00848=1093.463,435.135,396.354,178.711,25.327,153.886
C00849=1093.470,435.380,396.311,178.714,25.339,153.889
C00850=1093.476,435.626,396.268,178.717,25.351,153.891
C00851=1093.482,435.873,396.225,178.720,25.363,153.894
C00852=1093.489,436.119,396.182,178.723,25.375,153.897
C00853=1093.495,436.365,396.139,178.726,25.387,153.899
C00854=1093.502,436.611,396.095,178.729,25.399,153.902
C00855=1093.508,436.857,396.053,178.732,25.412,153.905
C00856=1093.514,437.103,396.009,178.735,25.424,153.907
C00857=1093.521,437.349,395.966,178.738,25.436,153.910
C00858=1093.528,437.595,395.923,178.742,25.449,153.913
C00859=1093.533,437.815,395.884,178.744,25.460,153.915
C00860=1093.539,438.034,395.846,178.747,25.471,153.918
C00861=1093.545,438.253,395.807,178.750,25.482,153.920
C00862=1093.551,438.472,395.768,178.753,25.493,153.923
C00863=1093.557,438.692,395.729,178.755,25.504,153.925
C00864=1093.562,438.910,395.691,178.758,25.516,153.928
C00865=1093.568,439.131,395.652,178.761,25.527,153.930
C00866=1093.574,439.350,395.614,178.764,25.538,153.933
C00867=1093.580,439.596,395.570,178.766,25.550,153.936
C00868=1093.587,439.842,395.526,178.770,25.564,153.938
C00869=1093.594,440.088,395.483,178.773,25.576,153.941
C00870=1093.600,440.334,395.439,178.776,25.589,153.944
C00871=1093.606,440.580,395.396,178.779,25.602,153.947
C00872=1093.613,440.826,395.352,178.782,25.615,153.950
C00873=1093.619,441.072,395.308,178.786,25.628,153.953
C00874=1093.626,441.318,395.265,178.788,25.641,153.956
C00875=1093.633,441.564,395.221,178.791,25.654,153.959
C00876=1093.639,441.810,395.177,178.795,25.668,153.962
C00877=1093.646,442.056,395.133,178.797,25.680,153.965
C00878=1093.652,442.302,395.089,178.800,25.694,153.968
C00879=1093.658,442.548,395.045,178.804,25.707,153.971
C00880=1093.665,442.793,395.001,178.807,25.721,153.974
C00881=1093.672,443.039,394.957,178.810,25.734,153.977
C00882=1093.678,443.285,394.913,178.813,25.747,153.980
C00883=1093.684,443.531,394.869,178.816,25.761,153.983
C00884=1093.691,443.776,394.825,178.819,25.774,153.986
C00885=1093.698,444.023,394.780,178.822,25.788,153.989
C00886=1093.705,444.269,394.737,178.826,25.802,153.992
C00887=1093.711,444.515,394.693,178.828,25.815,153.995
C00888=1093.717,444.760,394.648,178.830,25.829,153.998
C00889=1093.723,445.006,394.604,178.834,25.843,154.002
C00890=1093.730,445.252,394.559,178.835,25.856,154.005
C00891=1093.737,445.498,394.515,178.837,25.870,154.008
C00892=1093.744,445.744,394.470,178.840,25.883,154.011
C00893=1093.750,445.990,394.427,178.841,25.897,154.014
C00894=1093.756,446.235,394.381,178.843,25.910,154.018
C00895=1093.763,446.481,394.338,178.844,25.924,154.021
C00896=1093.769,446.727,394.293,178.846,25.938,154.024
C00897=1093.776,446.973,394.249,178.846,25.951,154.027
C00898=1093.782,447.219,394.204,178.847,25.964,154.031
C00899=1093.789,447.465,394.160,178.848,25.978,154.034
C00900=1093.796,447.711,394.115,178.849,25.992,154.037
C00901=1093.803,447.956,394.070,178.849,26.005,154.041
C00902=1093.809,448.203,394.026,178.850,26.019,154.044
C00903=1093.815,448.448,393.981,178.850,26.032,154.048
C00904=1093.823,448.694,393.936,178.850,26.045,154.051
C00905=1093.829,448.940,393.891,178.850,26.059,154.054
C00906=1093.835,449.186,393.847,178.849,26.072,154.058
C00907=1093.842,449.431,393.803,178.850,26.086,154.061
C00908=1093.849,449.677,393.758,178.849,26.099,154.065
C00909=1093.856,449.923,393.713,178.849,26.112,154.068
C00910=1093.864,450.168,393.669,178.848,26.124,154.071
C00911=1093.476,450.161,393.495,178.797,26.330,154.129
C00912=1093.467,449.914,393.539,178.797,26.318,154.126
C00913=1093.461,449.669,393.584,178.798,26.304,154.123
C00914=1093.454,449.424,393.629,178.798,26.291,154.119
C00915=1093.448,449.178,393.674,178.799,26.278,154.116
C00916=1093.441,448.931,393.718,178.798,26.264,154.112
C00917=1093.434,448.686,393.763,178.799,26.251,154.109
C00918=1093.428,448.440,393.808,178.798,26.237,154.105
C00919=1093.421,448.194,393.853,178.798,26.224,154.102
C00920=1093.414,447.949,393.897,178.797,26.210,154.099
C00921=1093.408,447.703,393.941,178.797,26.197,154.095
C00922=1093.401,447.456,393.987,178.796,26.183,154.092
C00923=1093.394,447.211,394.031,178.796,26.170,154.089
C00924=1093.388,446.965,394.075,178.794,26.156,154.085
C00925=1093.382,446.719,394.120,178.793,26.143,154.082
C00926=1093.375,446.473,394.165,178.792,26.129,154.079
C00927=1093.368,446.227,394.209,178.790,26.115,154.076
C00928=1093.361,445.982,394.253,178.789,26.102,154.072
C00929=1093.356,445.736,394.298,178.786,26.088,154.069
C00930=1093.348,445.490,394.343,178.785,26.075,154.066
C00931=1093.342,445.244,394.387,178.783,26.061,154.063
C00932=1093.335,444.998,394.431,178.780,26.047,154.059
C00933=1093.329,444.753,394.476,178.778,26.034,154.056
C00934=1093.322,444.506,394.520,178.775,26.020,154.053
C00935=1093.315,444.260,394.564,178.772,26.006,154.050
C00936=1093.308,444.015,394.608,178.769,25.992,154.047
C00937=1093.303,443.769,394.653,178.765,25.979,154.044
C00938=1093.296,443.523,394.697,178.763,25.965,154.041
C00939=1093.290,443.277,394.741,178.759,25.952,154.038
C00940=1093.283,443.031,394.785,178.756,25.938,154.034
C00941=1093.277,442.786,394.829,178.753,25.925,154.031
C00942=1093.270,442.540,394.874,178.749,25.911,154.028
C00943=1093.264,442.294,394.917,178.747,25.898,154.025
C00944=1093.256,442.048,394.962,178.743,25.885,154.022
C00945=1093.250,441.802,395.006,178.740,25.872,154.019
C00946=1093.244,441.556,395.049,178.738,25.858,154.016
C00947=1093.236,441.310,395.093,178.734,25.845,154.013
C00948=1093.230,441.064,395.136,178.731,25.832,154.011
C00949=1093.224,440.818,395.180,178.727,25.819,154.008
C00950=1093.217,440.572,395.224,178.725,25.806,154.005
C00951=1093.211,440.326,395.268,178.721,25.793,154.002
C00952=1093.204,440.080,395.312,178.718,25.780,153.999
C00953=1093.198,439.834,395.356,178.715,25.767,153.996
C00954=1093.191,439.588,395.399,178.712,25.754,153.993
C00955=1093.184,439.342,395.443,178.708,25.741,153.990
C00956=1093.179,439.128,395.480,178.706,25.731,153.988
C00957=1093.173,438.914,395.519,178.703,25.719,153.985
C00958=1093.167,438.700,395.557,178.700,25.709,153.983
C00959=1093.162,438.486,395.594,178.697,25.697,153.980
C00960=1093.156,438.273,395.632,178.695,25.687,153.978
C00961=1093.150,438.059,395.669,178.692,25.676,153.976
C00962=1093.145,437.845,395.707,178.689,25.665,153.973
C00963=1093.139,437.631,395.745,178.686,25.654,153.971
C00964=1093.132,437.385,395.788,178.684,25.642,153.968
C00965=1093.126,437.139,395.831,178.680,25.629,153.965
C00966=1093.120,436.893,395.875,178.678,25.617,153.963
C00967=1093.113,436.648,395.918,178.674,25.604,153.960
C00968=1093.107,436.401,395.961,178.671,25.592,153.957
C00969=1093.101,436.155,396.005,178.668,25.580,153.955
C00970=1093.094,435.909,396.048,178.665,25.568,153.952
C00971=1093.088,435.662,396.091,178.661,25.556,153.949
C00972=1093.080,435.417,396.134,178.659,25.544,153.947
C00973=1093.075,435.171,396.177,178.655,25.532,153.944
C00974=1093.069,434.925,396.221,178.653,25.520,153.941
C00975=1093.062,434.678,396.263,178.649,25.508,153.939
C00976=1093.056,434.432,396.306,178.646,25.496,153.936
C00977=1093.049,434.186,396.349,178.643,25.484,153.933
C00978=1093.043,433.940,396.392,178.640,25.472,153.931
C00979=1093.036,433.694,396.435,178.636,25.460,153.928
C00980=1093.030,433.447,396.478,178.634,25.449,153.926
C00981=1093.024,433.201,396.521,178.630,25.436,153.923
C00982=1093.018,432.955,396.563,178.627,25.425,153.920
C00983=1093.011,432.709,396.606,178.624,25.414,153.918
C00984=1093.005,432.463,396.649,178.621,25.402,153.915
C00985=1092.998,432.217,396.691,178.618,25.390,153.913
C00986=1092.991,431.970,396.734,178.615,25.379,153.910
C00987=1092.985,431.724,396.777,178.612,25.367,153.908
C00988=1092.979,431.478,396.819,178.609,25.356,153.905
C00989=1092.972,431.232,396.862,178.605,25.344,153.903
C00990=1092.966,430.985,396.905,178.602,25.333,153.901
C00991=1092.960,430.740,396.947,178.599,25.322,153.898
C00992=1092.953,430.493,396.989,178.596,25.311,153.896
C00993=1092.947,430.247,397.033,178.593,25.299,153.893
C00994=1092.941,430.001,397.074,178.590,25.288,153.891
C00995=1092.934,429.754,397.117,178.586,25.277,153.888
C00996=1092.929,429.509,397.159,178.584,25.266,153.886
C00997=1092.922,429.262,397.202,178.581,25.255,153.884
C00998=1092.916,429.016,397.243,178.578,25.244,153.881
C00999=1092.909,428.770,397.286,178.574,25.232,153.879
C01000=1092.902,428.523,397.328,178.571,25.222,153.877
C01001=1092.897,428.277,397.370,178.568,25.211,153.874
C01002=1092.890,428.031,397.413,178.565,25.200,153.872
C01003=1092.884,427.784,397.454,178.562,25.189,153.869
C01004=1092.877,427.538,397.497,178.559,25.178,153.867
C01005=1092.871,427.291,397.539,178.556,25.168,153.865
C01006=1092.864,427.046,397.581,178.553,25.157,153.863
C01007=1092.858,426.799,397.623,178.550,25.147,153.860
C01008=1092.852,426.553,397.665,178.546,25.135,153.858
C01009=1092.845,426.306,397.707,178.543,25.125,153.856
C01010=1092.839,426.061,397.749,178.540,25.115,153.854
C01011=1092.832,425.814,397.791,178.537,25.104,153.851
C01012=1092.827,425.584,397.830,178.534,25.094,153.849
C01013=1092.821,425.354,397.870,178.531,25.084,153.847
C01014=1092.815,425.123,397.908,178.529,25.075,153.845
C01015=1092.809,424.892,397.947,178.526,25.065,153.843
C01016=1092.803,424.663,397.986,178.523,25.055,153.841
C01017=1092.797,424.433,398.026,178.520,25.045,153.839
C01018=1092.791,424.202,398.064,178.517,25.036,153.837
C01019=1092.786,423.972,398.103,178.514,25.026,153.835
C01020=1092.779,423.725,398.145,178.511,25.016,153.833
C01021=1092.773,423.479,398.186,178.508,25.006,153.830
C01022=1092.767,423.232,398.228,178.505,24.995,153.828
C01023=1092.761,422.986,398.270,178.502,24.985,153.826
C01024=1092.755,422.740,398.311,178.499,24.975,153.824
C01025=1092.748,422.493,398.353,178.495,24.965,153.822
C01026=1092.742,422.247,398.394,178.492,24.955,153.820
C01027=1092.735,422.000,398.436,178.489,24.945,153.818
C01028=1092.729,421.754,398.477,178.486,24.935,153.816
C01029=1092.723,421.508,398.519,178.483,24.925,153.814
C01030=1092.717,421.261,398.560,178.480,24.915,153.812
C01031=1092.710,421.015,398.601,178.477,24.905,153.809
C01032=1092.704,420.769,398.643,178.474,24.895,153.807
C01033=1092.698,420.522,398.684,178.471,24.885,153.805
C01034=1092.692,420.275,398.725,178.468,24.876,153.803
C01035=1092.685,420.029,398.766,178.465,24.866,153.801
C01036=1092.679,419.782,398.808,178.461,24.856,153.799
C01037=1092.673,419.536,398.849,178.458,24.846,153.797
C01038=1092.666,419.289,398.890,178.455,24.837,153.795
C01039=1092.660,419.043,398.931,178.453,24.827,153.793
C01040=1092.654,418.796,398.973,178.450,24.818,153.791
C01041=1092.647,418.550,399.013,178.447,24.808,153.789
C01042=1092.642,418.304,399.054,178.444,24.799,153.787
C01043=1092.636,418.057,399.095,178.441,24.789,153.785
C01044=1092.629,417.810,399.136,178.437,24.780,153.783
C01045=1092.623,417.563,399.177,178.434,24.770,153.781
C01046=1092.617,417.317,399.219,178.431,24.761,153.780
C01047=1092.611,417.071,399.259,178.428,24.751,153.778
C01048=1092.605,416.824,399.300,178.425,24.742,153.776
C01049=1092.599,416.578,399.341,178.423,24.732,153.774
C01050=1092.592,416.331,399.382,178.419,24.723,153.772
C01051=1092.586,416.084,399.423,178.416,24.714,153.770
C01052=1092.580,415.838,399.463,178.413,24.705,153.768
C01053=1092.573,415.592,399.504,178.410,24.695,153.766
C01054=1092.567,415.345,399.545,178.406,24.686,153.764
C01055=1092.560,415.098,399.585,178.404,24.678,153.762
C01056=1092.555,414.851,399.626,178.401,24.668,153.761
C01057=1092.548,414.605,399.667,178.398,24.659,153.759
C01058=1092.542,414.358,399.707,178.394,24.650,153.757
C01059=1092.536,414.112,399.748,178.391,24.641,153.755
C01060=1092.530,413.865,399.788,178.389,24.632,153.753
C01061=1092.523,413.619,399.828,178.386,24.623,153.751
C01062=1092.517,413.371,399.869,178.382,24.614,153.750
C01063=1092.510,413.125,399.910,178.379,24.605,153.748
C01064=1092.505,412.878,399.951,178.377,24.597,153.746
C01065=1092.498,412.632,399.991,178.373,24.588,153.744
C01066=1092.492,412.385,400.031,178.370,24.579,153.743
C01067=1092.486,412.139,400.071,178.368,24.570,153.741
C01068=1092.480,411.916,400.108,178.364,24.562,153.739
C01069=1092.474,411.693,400.144,178.362,24.554,153.738
C01070=1092.469,411.470,400.180,178.359,24.546,153.736
C01071=1092.464,411.247,400.216,178.357,24.538,153.734
C01072=1092.458,411.024,400.253,178.354,24.530,153.733
C01073=1092.453,410.801,400.290,178.351,24.523,153.731
C01074=1092.447,410.578,400.326,178.349,24.515,153.730
C01075=1092.441,410.355,400.363,178.345,24.507,153.728
C01076=1092.435,410.108,400.402,178.343,24.498,153.726
C01077=1092.430,409.862,400.442,178.340,24.490,153.725
C01078=1092.424,409.615,400.483,178.337,24.482,153.723
C01079=1092.417,409.369,400.523,178.334,24.473,153.721
C01080=1092.411,409.122,400.562,178.330,24.464,153.720
C01081=1092.405,408.875,400.602,178.328,24.456,153.718
C01082=1092.399,408.629,400.643,178.325,24.447,153.716
C01083=1092.393,408.381,400.683,178.321,24.438,153.714
C01084=1092.387,408.135,400.723,178.319,24.430,153.713
C01085=1092.381,407.888,400.763,178.315,24.422,153.711
C01086=1092.374,407.641,400.802,178.313,24.414,153.710
C01087=1092.368,407.395,400.842,178.309,24.406,153.708
C01088=1092.363,407.148,400.882,178.307,24.397,153.706
C01089=1092.356,406.902,400.922,178.304,24.389,153.705
C01090=1092.350,406.654,400.961,178.301,24.381,153.703
C01091=1092.344,406.408,401.001,178.298,24.373,153.701
C01092=1092.338,406.160,401.041,178.294,24.364,153.700
C01093=1092.332,405.914,401.081,178.292,24.356,153.698
C01094=1092.326,405.667,401.121,178.288,24.348,153.697
C01095=1092.320,405.421,401.161,178.286,24.340,153.695
C01096=1092.313,405.174,401.200,178.282,24.332,153.693
C01097=1092.307,404.927,401.239,178.280,24.324,153.692
C01098=1092.301,404.681,401.279,178.276,24.316,153.690
C01099=1092.295,404.433,401.319,178.274,24.308,153.689
C01100=1092.289,404.186,401.358,178.271,24.300,153.687
C01101=1092.283,403.940,401.398,178.268,24.292,153.686
C01102=1092.277,403.693,401.437,178.265,24.284,153.684
C01103=1092.271,403.446,401.477,178.262,24.276,153.682
C01104=1092.265,403.199,401.516,178.259,24.268,153.681
C01105=1092.258,402.953,401.556,178.256,24.260,153.679
C01106=1092.252,402.706,401.595,178.253,24.253,153.678
C01107=1092.246,402.459,401.634,178.249,24.245,153.676
C01108=1092.240,402.212,401.674,178.247,24.237,153.675
C01109=1092.235,401.966,401.713,178.244,24.230,153.673
C01110=1092.228,401.719,401.751,178.241,24.222,153.672
C01111=1092.222,401.472,401.791,178.238,24.214,153.670
C01112=1092.216,401.225,401.830,178.235,24.206,153.669
C01113=1092.210,400.978,401.869,178.232,24.198,153.667
C01114=1092.204,400.731,401.909,178.229,24.191,153.666
C01115=1092.197,400.484,401.948,178.226,24.183,153.665
C01116=1092.192,400.238,401.987,178.223,24.176,153.663
C01117=1092.186,399.991,402.026,178.221,24.168,153.662
C01118=1092.180,399.743,402.066,178.217,24.160,153.660
C01119=1092.173,399.497,402.104,178.214,24.153,153.659
C01120=1092.167,399.250,402.143,178.212,24.146,153.657
C01121=1092.161,399.003,402.183,178.208,24.138,153.656
C01122=1092.155,398.757,402.221,178.205,24.130,153.654
C01123=1092.149,398.509,402.260,178.203,24.123,153.653
C01124=1092.144,398.288,402.296,178.200,24.116,153.652
C01125=1092.138,398.065,402.331,178.197,24.109,153.650
C01126=1092.133,397.842,402.365,178.194,24.103,153.649
C01127=1092.127,397.620,402.400,178.192,24.096,153.648
C01128=1092.122,397.397,402.435,178.189,24.090,153.647
C01129=1092.116,397.174,402.470,178.186,24.083,153.645
C01130=1092.111,396.952,402.505,178.183,24.076,153.644
C01131=1092.105,396.729,402.540,178.181,24.070,153.643
C01132=1092.100,396.483,402.579,178.178,24.062,153.642
C01133=1092.093,396.236,402.618,178.175,24.055,153.640
C01134=1092.088,395.989,402.656,178.172,24.048,153.639
C01135=1092.081,395.742,402.695,178.169,24.040,153.638
C01136=1092.076,395.495,402.734,178.166,24.034,153.636
C01137=1092.069,395.248,402.772,178.163,24.027,153.635
C01138=1092.064,395.001,402.811,178.160,24.019,153.634
C01139=1092.057,394.754,402.850,178.157,24.012,153.632
C01140=1092.051,394.508,402.887,178.154,24.005,153.631
C01141=1092.045,394.260,402.927,178.151,23.998,153.630
C01142=1092.039,394.014,402.965,178.148,23.991,153.628
C01143=1092.033,393.768,403.003,178.146,23.984,153.627
C01144=1092.027,393.520,403.042,178.142,23.977,153.626
C01145=1092.021,393.274,403.080,178.139,23.970,153.624
C01146=1092.015,393.026,403.119,178.136,23.963,153.623
C01147=1092.009,392.780,403.157,178.134,23.956,153.622
C01148=1092.002,392.532,403.195,178.131,23.949,153.620
C01149=1091.997,392.285,403.234,178.127,23.942,153.619
C01150=1091.991,392.039,403.272,178.124,23.935,153.618
C01151=1091.985,391.792,403.310,178.121,23.928,153.617
C01152=1091.979,391.545,403.348,178.119,23.922,153.615
C01153=1091.972,391.298,403.386,178.116,23.915,153.614
C01154=1091.967,391.051,403.425,178.112,23.908,153.613
C01155=1091.961,390.804,403.463,178.109,23.901,153.612
C01156=1091.954,390.557,403.501,178.106,23.894,153.611
C01157=1091.948,390.310,403.539,178.103,23.888,153.609
C01158=1091.942,390.063,403.577,178.101,23.881,153.608
C01159=1091.936,389.817,403.616,178.098,23.875,153.607
C01160=1091.930,389.570,403.653,178.094,23.867,153.606
C01161=1091.923,389.322,403.691,178.091,23.861,153.604
C01162=1091.917,389.076,403.729,178.088,23.854,153.603
C01163=1091.912,388.829,403.768,178.085,23.848,153.602
C01164=1091.906,388.582,403.805,178.082,23.841,153.601
C01165=1091.900,388.335,403.843,178.079,23.835,153.600
C01166=1091.894,388.088,403.881,178.077,23.828,153.599
C01167=1091.888,387.841,403.919,178.073,23.821,153.597
C01168=1091.882,387.594,403.957,178.070,23.814,153.596
C01169=1091.876,387.347,403.995,178.067,23.808,153.595
C01170=1091.870,387.100,404.033,178.064,23.801,153.594
C01171=1091.864,386.853,404.070,178.061,23.795,153.593
C01172=1091.858,386.607,404.108,178.058,23.788,153.591
C01173=1091.851,386.359,404.146,178.055,23.782,153.590
C01174=1091.846,386.112,404.183,178.052,23.776,153.589
C01175=1091.840,385.865,404.221,178.049,23.769,153.588
C01176=1091.834,385.618,404.259,178.046,23.763,153.587
C01177=1091.828,385.372,404.297,178.043,23.756,153.586
C01178=1091.822,385.125,404.334,178.040,23.749,153.585
C01179=1091.816,384.877,404.372,178.037,23.743,153.583
C01180=1091.811,384.661,404.405,178.035,23.737,153.582
C01181=1091.806,384.446,404.438,178.032,23.732,153.581
C01182=1091.801,384.229,404.470,178.029,23.726,153.581
C01183=1091.796,384.014,404.504,178.027,23.721,153.580
C01184=1091.791,383.797,404.536,178.024,23.715,153.579
C01185=1091.784,383.582,404.569,178.021,23.710,153.578
C01186=1091.780,383.366,404.601,178.018,23.704,153.577
C01187=1091.775,383.150,404.634,178.016,23.699,153.576
C01188=1091.769,382.903,404.672,178.013,23.692,153.575
C01189=1091.763,382.656,404.709,178.010,23.686,153.573
C01190=1091.757,382.409,404.747,178.007,23.680,153.572
C01191=1091.750,382.161,404.784,178.004,23.674,153.571
C01192=1091.744,381.915,404.821,178.001,23.667,153.570
C01193=1091.739,381.667,404.858,177.998,23.662,153.569
C01194=1091.733,381.421,404.896,177.995,23.655,153.568
C01195=1091.727,381.173,404.933,177.992,23.649,153.567
C01196=1091.721,380.927,404.970,177.989,23.643,153.566
C01197=1091.715,380.679,405.007,177.986,23.637,153.565
C01198=1091.709,380.433,405.045,177.983,23.631,153.564
C01199=1091.703,380.186,405.082,177.980,23.625,153.563
C01200=1091.697,379.937,405.119,177.977,23.619,153.562
C01201=1091.691,379.691,405.157,177.974,23.613,153.561
C01202=1091.684,379.444,405.193,177.971,23.607,153.560
C01203=1091.679,379.196,405.230,177.968,23.601,153.559
C01204=1091.673,378.950,405.268,177.965,23.595,153.558
C01205=1091.667,378.703,405.305,177.961,23.589,153.557
C01206=1091.661,378.455,405.342,177.958,23.582,153.556
C01207=1091.655,378.208,405.378,177.955,23.577,153.555
C01208=1091.649,377.961,405.416,177.952,23.571,153.554
C01209=1091.643,377.714,405.453,177.950,23.565,153.553
C01210=1091.637,377.467,405.489,177.947,23.559,153.552
C01211=1091.631,377.220,405.526,177.944,23.554,153.551
C01212=1091.626,376.972,405.563,177.941,23.547,153.550
C01213=1091.619,376.725,405.600,177.938,23.541,153.549
C01214=1091.614,376.478,405.637,177.935,23.535,153.548
C01215=1091.608,376.232,405.674,177.932,23.530,153.547
C01216=1091.602,375.985,405.711,177.929,23.524,153.546
C01217=1091.596,375.737,405.748,177.925,23.518,153.545
C01218=1091.590,375.490,405.784,177.922,23.512,153.544
C01219=1091.585,375.243,405.821,177.919,23.506,153.543
C01220=1091.578,374.996,405.858,177.916,23.501,153.542
C01221=1091.573,374.749,405.895,177.914,23.495,153.541
C01222=1091.566,374.501,405.931,177.911,23.489,153.540
C01223=1091.561,374.254,405.968,177.908,23.483,153.539
C01224=1091.555,374.006,406.004,177.905,23.477,153.538
C01225=1091.549,373.759,406.041,177.901,23.472,153.537
C01226=1091.543,373.512,406.077,177.898,23.466,153.536
C01227=1091.537,373.266,406.113,177.895,23.461,153.535
C01228=1091.531,373.018,406.150,177.892,23.455,153.534
C01229=1091.525,372.771,406.187,177.890,23.450,153.534
C01230=1091.519,372.524,406.223,177.886,23.444,153.533
C01231=1091.513,372.276,406.260,177.883,23.438,153.532
C01232=1091.507,372.029,406.296,177.880,23.433,153.531
C01233=1091.501,371.782,406.333,177.877,23.427,153.530
C01234=1091.495,371.535,406.370,177.874,23.421,153.529
C01235=1091.489,371.287,406.405,177.871,23.416,153.528
C01236=1091.480,370.883,406.465,177.866,23.407,153.527
C01237=1091.470,370.479,406.524,177.861,23.398,153.525
C01238=1091.460,370.075,406.583,177.856,23.389,153.524
C01239=1091.450,369.670,406.643,177.851,23.380,153.522
C01240=1091.445,369.424,406.679,177.848,23.374,153.521
C01241=1091.439,369.176,406.715,177.845,23.369,153.521
C01242=1091.433,368.929,406.751,177.842,23.364,153.520
C01243=1091.427,368.681,406.787,177.839,23.359,153.519
C01244=1091.421,368.434,406.824,177.836,23.353,153.518
C01245=1091.415,368.187,406.859,177.833,23.348,153.517
C01246=1091.410,367.940,406.896,177.829,23.342,153.516
C01247=1091.404,367.692,406.932,177.827,23.337,153.515
C01248=1091.398,367.446,406.968,177.824,23.331,153.515
C01249=1091.392,367.198,407.003,177.821,23.326,153.514
C01250=1091.386,366.951,407.040,177.818,23.320,153.513
C01251=1091.380,366.703,407.076,177.814,23.315,153.512
C01252=1091.375,366.456,407.112,177.812,23.310,153.511
C01253=1091.368,366.209,407.148,177.809,23.305,153.510
C01254=1091.362,365.961,407.184,177.805,23.299,153.510
C01255=1091.357,365.714,407.219,177.802,23.294,153.509
C01256=1091.351,365.467,407.256,177.800,23.289,153.508
C01257=1091.345,365.220,407.291,177.797,23.284,153.507
C01258=1091.339,364.973,407.327,177.793,23.279,153.506
C01259=1091.333,364.725,407.362,177.790,23.273,153.505
C01260=1091.327,364.477,407.398,177.788,23.268,153.505
C01261=1091.321,364.230,407.435,177.784,23.263,153.504
C01262=1091.315,363.983,407.470,177.781,23.258,153.503
C01263=1091.309,363.736,407.506,177.778,23.253,153.502
C01264=1091.303,363.488,407.541,177.775,23.248,153.501
C01265=1091.298,363.241,407.577,177.772,23.243,153.501
C01266=1091.292,362.993,407.613,177.769,23.237,153.500
C01267=1091.286,362.746,407.648,177.765,23.232,153.499
C01268=1091.280,362.499,407.684,177.763,23.227,153.498
C01269=1091.274,362.251,407.719,177.760,23.222,153.498
C01270=1091.269,362.005,407.755,177.756,23.217,153.497
C01271=1091.263,361.757,407.791,177.754,23.212,153.496
C01272=1091.257,361.509,407.827,177.751,23.207,153.495
C01273=1091.251,361.262,407.862,177.747,23.202,153.495
C01274=1091.245,361.014,407.897,177.745,23.197,153.494
C01275=1091.239,360.767,407.932,177.742,23.191,153.493
C01276=1091.233,360.520,407.968,177.738,23.186,153.492
C01277=1091.227,360.272,408.003,177.735,23.181,153.492
C01278=1091.222,360.025,408.039,177.732,23.177,153.491
C01279=1091.216,359.777,408.075,177.729,23.171,153.490
C01280=1091.210,359.531,408.109,177.726,23.166,153.489
C01281=1091.204,359.283,408.145,177.723,23.162,153.489
C01282=1091.198,359.035,408.180,177.720,23.157,153.488
C01283=1091.192,358.788,408.215,177.717,23.152,153.487
C01284=1091.186,358.540,408.251,177.714,23.147,153.486
C01285=1091.180,358.293,408.286,177.711,23.142,153.486
C01286=1091.174,358.045,408.321,177.707,23.137,153.485
C01287=1091.169,357.798,408.356,177.705,23.133,153.484
C01288=1091.159,357.410,408.412,177.700,23.124,153.483
C01289=1091.150,357.021,408.467,177.695,23.117,153.482
C01290=1091.141,356.631,408.522,177.690,23.110,153.481
C01291=1091.132,356.243,408.577,177.686,23.102,153.480
C01292=1091.125,355.995,408.612,177.683,23.097,153.479
C01293=1091.120,355.748,408.647,177.679,23.092,153.478
C01294=1091.114,355.500,408.682,177.677,23.088,153.478
C01295=1091.108,355.253,408.717,177.673,23.083,153.477
C01296=1091.102,355.005,408.752,177.670,23.078,153.476
C01297=1091.097,354.758,408.787,177.667,23.073,153.476
C01298=1091.090,354.510,408.822,177.664,23.068,153.475
C01299=1091.085,354.263,408.857,177.661,23.064,153.474
C01300=1091.080,354.015,408.892,177.658,23.059,153.474
C01301=1091.073,353.768,408.927,177.655,23.054,153.473
C01302=1091.068,353.520,408.962,177.652,23.049,153.472
C01303=1091.062,353.272,408.996,177.649,23.045,153.472
C01304=1091.056,353.026,409.031,177.646,23.040,153.471
C01305=1091.050,352.778,409.065,177.643,23.036,153.470
C01306=1091.044,352.531,409.101,177.639,23.031,153.470
C01307=1091.038,352.283,409.135,177.637,23.026,153.469
C01308=1091.033,352.035,409.170,177.633,23.021,153.468
C01309=1091.027,351.788,409.204,177.631,23.017,153.468
C01310=1091.021,351.540,409.240,177.627,23.012,153.467
C01311=1091.015,351.293,409.274,177.624,23.008,153.466
C01312=1091.009,351.045,409.308,177.621,23.003,153.466
C01313=1091.003,350.797,409.343,177.618,22.999,153.465
C01314=1090.997,350.551,409.378,177.615,22.994,153.464
C01315=1090.992,350.303,409.413,177.612,22.989,153.464
C01316=1090.986,350.055,409.447,177.609,22.985,153.463
C01317=1090.980,349.808,409.481,177.606,22.980,153.463
C01318=1090.975,349.560,409.516,177.603,22.976,153.462
C01319=1090.968,349.313,409.551,177.600,22.971,153.461
C01320=1090.963,349.065,409.585,177.596,22.966,153.461
C01321=1090.957,348.818,409.620,177.594,22.962,153.460
C01322=1090.950,348.570,409.654,177.590,22.957,153.459
C01323=1090.945,348.322,409.689,177.588,22.953,153.459
C01324=1090.939,348.075,409.723,177.584,22.949,153.458
C01325=1090.933,347.827,409.757,177.582,22.944,153.458
C01326=1090.928,347.579,409.792,177.578,22.939,153.457
C01327=1090.922,347.332,409.826,177.576,22.935,153.456
C01328=1090.916,347.085,409.860,177.572,22.931,153.456
C01329=1090.910,346.837,409.894,177.569,22.927,153.455
C01330=1090.905,346.589,409.929,177.566,22.922,153.455
C01331=1090.899,346.342,409.963,177.563,22.918,153.454
C01332=1090.893,346.095,409.997,177.560,22.913,153.453
C01333=1090.887,345.846,410.032,177.557,22.909,153.453
C01334=1090.882,345.598,410.065,177.554,22.904,153.452
C01335=1090.876,345.351,410.099,177.551,22.900,153.452
C01336=1090.870,345.104,410.133,177.548,22.895,153.451
C01337=1090.863,344.856,410.168,177.545,22.891,153.450
C01338=1090.858,344.608,410.203,177.541,22.887,153.450
C01339=1090.853,344.360,410.236,177.539,22.882,153.449
C01340=1090.843,343.975,410.289,177.534,22.876,153.449
C01341=1090.834,343.588,410.342,177.529,22.869,153.448
C01342=1090.824,343.202,410.396,177.524,22.862,153.447
C01343=1090.816,342.816,410.448,177.520,22.856,153.446
C01344=1090.810,342.568,410.483,177.516,22.851,153.445
C01345=1090.804,342.320,410.516,177.513,22.847,153.445
C01346=1090.798,342.073,410.550,177.510,22.842,153.444
C01347=1090.793,341.825,410.583,177.507,22.839,153.444
C01348=1090.787,341.578,410.617,177.504,22.834,153.443
C01349=1090.781,341.330,410.651,177.501,22.830,153.443
C01350=1090.775,341.082,410.685,177.498,22.826,153.442
C01351=1090.769,340.834,410.719,177.495,22.821,153.441
C01352=1090.763,340.586,410.753,177.492,22.818,153.441
C01353=1090.758,340.339,410.787,177.489,22.813,153.440
C01354=1090.752,340.091,410.820,177.486,22.809,153.440
C01355=1090.746,339.844,410.854,177.482,22.805,153.439
C01356=1090.741,339.596,410.887,177.480,22.800,153.439
C01357=1090.735,339.349,410.921,177.476,22.796,153.438
C01358=1090.729,339.101,410.955,177.473,22.792,153.438
C01359=1090.723,338.854,410.989,177.471,22.788,153.437
C01360=1090.718,338.606,411.022,177.467,22.783,153.437
C01361=1090.712,338.358,411.055,177.464,22.780,153.436
C01362=1090.706,338.110,411.090,177.461,22.775,153.436
C01363=1090.699,337.862,411.123,177.458,22.771,153.435
C01364=1090.694,337.614,411.156,177.456,22.767,153.435
C01365=1090.688,337.367,411.190,177.452,22.763,153.434
C01366=1090.683,337.119,411.223,177.449,22.759,153.434
C01367=1090.677,336.871,411.257,177.446,22.755,153.433
C01368=1090.671,336.624,411.291,177.443,22.751,153.432
C01369=1090.665,336.376,411.323,177.440,22.747,153.432
C01370=1090.659,336.128,411.357,177.437,22.743,153.432
C01371=1090.654,335.881,411.390,177.434,22.739,153.431
C01372=1090.648,335.633,411.424,177.430,22.735,153.431
C01373=1090.642,335.386,411.457,177.428,22.730,153.430
C01374=1090.636,335.138,411.490,177.425,22.727,153.430
C01375=1090.630,334.890,411.524,177.421,22.723,153.429
C01376=1090.625,334.642,411.557,177.419,22.718,153.429
C01377=1090.619,334.394,411.590,177.416,22.715,153.428
C01378=1090.613,334.146,411.623,177.412,22.711,153.428
C01379=1090.607,333.899,411.657,177.409,22.706,153.427
C01380=1090.602,333.651,411.690,177.406,22.702,153.427
C01381=1090.595,333.404,411.723,177.403,22.699,153.426
C01382=1090.590,333.156,411.756,177.400,22.695,153.426
C01383=1090.584,332.908,411.790,177.397,22.690,153.425
C01384=1090.578,332.660,411.823,177.394,22.687,153.425
C01385=1090.572,332.412,411.856,177.391,22.683,153.424
C01386=1090.567,332.164,411.889,177.388,22.678,153.424
C01387=1090.561,331.917,411.922,177.385,22.675,153.423
C01388=1090.556,331.670,411.955,177.382,22.671,153.423
C01389=1090.549,331.422,411.988,177.378,22.667,153.422
C01390=1090.544,331.174,412.021,177.376,22.663,153.422
C01391=1090.538,330.926,412.053,177.373,22.659,153.421
C01392=1090.528,330.534,412.106,177.368,22.653,153.421
C01393=1090.519,330.142,412.158,177.363,22.647,153.420
C01394=1090.509,329.750,412.210,177.358,22.641,153.420
C01395=1090.500,329.357,412.262,177.353,22.635,153.419
C01396=1090.495,329.110,412.294,177.350,22.631,153.418
C01397=1090.489,328.862,412.327,177.347,22.627,153.418
C01398=1090.483,328.614,412.360,177.343,22.624,153.418
C01399=1090.476,328.367,412.393,177.341,22.620,153.417
C01400=1090.471,328.118,412.426,177.338,22.616,153.417
C01401=1090.465,327.870,412.458,177.335,22.613,153.416
C01402=1090.459,327.623,412.491,177.331,22.608,153.416
C01403=1090.453,327.374,412.524,177.329,22.605,153.415
C01404=1090.448,327.127,412.556,177.326,22.601,153.415
C01405=1090.442,326.880,412.589,177.322,22.597,153.414
C01406=1090.436,326.631,412.621,177.319,22.594,153.414
C01407=1090.430,326.384,412.654,177.317,22.590,153.414
C01408=1090.424,326.136,412.688,177.314,22.586,153.413
C01409=1090.418,325.888,412.720,177.310,22.582,153.413
C01410=1090.413,325.641,412.752,177.307,22.578,153.412
C01411=1090.407,325.392,412.785,177.304,22.575,153.412
C01412=1090.401,325.145,412.817,177.302,22.571,153.412
C01413=1090.395,324.896,412.849,177.298,22.567,153.411
C01414=1090.389,324.649,412.882,177.295,22.563,153.411
C01415=1090.384,324.401,412.914,177.292,22.560,153.410
C01416=1090.378,324.153,412.947,177.289,22.556,153.410
C01417=1090.372,323.905,412.979,177.286,22.552,153.410
C01418=1090.367,323.658,413.012,177.283,22.549,153.409
C01419=1090.361,323.410,413.044,177.280,22.545,153.409
C01420=1090.355,323.162,413.077,177.277,22.542,153.408
C01421=1090.349,322.914,413.109,177.274,22.538,153.408
C01422=1090.344,322.666,413.141,177.271,22.534,153.407
C01423=1090.338,322.419,413.174,177.268,22.531,153.407
C01424=1090.332,322.170,413.206,177.265,22.527,153.407
C01425=1090.326,321.923,413.238,177.261,22.523,153.406
C01426=1090.321,321.675,413.271,177.259,22.519,153.406
C01427=1090.315,321.427,413.303,177.256,22.516,153.406
C01428=1090.309,321.179,413.335,177.253,22.512,153.405
C01429=1090.303,320.932,413.367,177.249,22.508,153.405
C01430=1090.297,320.683,413.399,177.246,22.505,153.404
C01431=1090.292,320.436,413.432,177.244,22.501,153.404
C01432=1090.286,320.187,413.464,177.241,22.498,153.404
C01433=1090.281,319.940,413.496,177.238,22.494,153.403
C01434=1090.275,319.692,413.528,177.234,22.490,153.403
C01435=1090.269,319.444,413.560,177.231,22.486,153.402
C01436=1090.264,319.196,413.592,177.229,22.483,153.402
C01437=1090.258,318.948,413.624,177.226,22.479,153.402
C01438=1090.253,318.700,413.656,177.223,22.476,153.401
C01439=1090.247,318.453,413.689,177.219,22.472,153.401
C01440=1090.241,318.205,413.721,177.216,22.468,153.400
C01441=1090.235,317.957,413.752,177.213,22.465,153.400
C01442=1090.229,317.709,413.784,177.211,22.461,153.400
C01443=1090.225,317.461,413.817,177.208,22.458,153.399
C01444=1090.215,317.062,413.867,177.203,22.452,153.399
C01445=1090.206,316.663,413.919,177.198,22.446,153.398
C01446=1090.197,316.264,413.970,177.193,22.440,153.397
C01447=1090.188,315.865,414.021,177.188,22.434,153.397
C01448=1090.182,315.617,414.053,177.185,22.431,153.397
C01449=1090.177,315.369,414.085,177.182,22.427,153.396
C01450=1090.171,315.121,414.117,177.179,22.424,153.396
C01451=1090.165,314.873,414.149,177.176,22.420,153.395
C01452=1090.159,314.625,414.181,177.173,22.417,153.395
C01453=1090.154,314.378,414.213,177.170,22.413,153.395
C01454=1090.147,314.130,414.244,177.166,22.410,153.394
C01455=1090.142,313.882,414.276,177.163,22.406,153.394
C01456=1090.136,313.634,414.308,177.160,22.403,153.394
C01457=1090.131,313.386,414.339,177.158,22.400,153.393
C01458=1090.124,313.138,414.370,177.155,22.396,153.393
C01459=1090.118,312.890,414.402,177.152,22.393,153.393
C01460=1090.113,312.642,414.434,177.149,22.390,153.392
C01461=1090.106,312.394,414.464,177.145,22.386,153.392
C01462=1090.101,312.146,414.496,177.142,22.383,153.392
C01463=1090.095,311.898,414.528,177.139,22.379,153.392
C01464=1090.089,311.651,414.559,177.136,22.376,153.391
C01465=1090.083,311.402,414.590,177.133,22.373,153.391
C01466=1090.078,311.154,414.622,177.131,22.369,153.390
C01467=1090.072,310.907,414.653,177.128,22.366,153.390
C01468=1090.066,310.658,414.685,177.124,22.362,153.390
C01469=1090.061,310.411,414.716,177.121,22.359,153.390
C01470=1090.054,310.163,414.748,177.118,22.356,153.389
C01471=1090.049,309.915,414.779,177.115,22.352,153.389
C01472=1090.043,309.667,414.811,177.112,22.349,153.389
C01473=1090.037,309.419,414.842,177.109,22.346,153.388
C01474=1090.032,309.171,414.873,177.106,22.343,153.388
C01475=1090.026,308.923,414.905,177.103,22.339,153.388
C01476=1090.020,308.675,414.935,177.099,22.336,153.387
C01477=1090.014,308.427,414.967,177.096,22.332,153.387
C01478=1090.008,308.179,414.997,177.094,22.329,153.387
C01479=1090.003,307.932,415.029,177.091,22.326,153.387
C01480=1089.997,307.683,415.060,177.088,22.323,153.386
C01481=1089.991,307.436,415.091,177.085,22.319,153.386
C01482=1089.986,307.188,415.122,177.082,22.316,153.385
C01483=1089.979,306.940,415.154,177.079,22.312,153.385
C01484=1089.974,306.692,415.185,177.075,22.309,153.385
C01485=1089.968,306.444,415.215,177.072,22.305,153.385
C01486=1089.963,306.196,415.247,177.069,22.302,153.384
C01487=1089.956,305.948,415.277,177.066,22.299,153.384
C01488=1089.951,305.700,415.309,177.063,22.296,153.384
C01489=1089.945,305.452,415.339,177.061,22.292,153.383
C01490=1089.939,305.203,415.371,177.058,22.289,153.383
C01491=1089.934,304.956,415.402,177.055,22.286,153.383
C01492=1089.928,304.708,415.433,177.052,22.283,153.382
C01493=1089.923,304.460,415.464,177.049,22.280,153.382
C01494=1089.916,304.212,415.495,177.045,22.276,153.382
C01495=1089.911,303.964,415.526,177.042,22.273,153.382
C01496=1089.902,303.568,415.574,177.038,22.268,153.381
C01497=1089.893,303.172,415.625,177.032,22.262,153.381
C01498=1089.884,302.775,415.674,177.028,22.257,153.380
C01499=1089.875,302.379,415.723,177.023,22.252,153.380
C01500=1089.870,302.131,415.753,177.020,22.248,153.379
C01501=1089.864,301.883,415.785,177.017,22.245,153.379
C01502=1089.858,301.635,415.816,177.014,22.242,153.379
C01503=1089.852,301.387,415.846,177.011,22.239,153.379
C01504=1089.847,301.139,415.877,177.008,22.235,153.378
C01505=1089.841,300.891,415.907,177.005,22.232,153.378
C01506=1089.836,300.643,415.938,177.002,22.229,153.378
C01507=1089.830,300.395,415.968,176.999,22.226,153.377
C01508=1089.825,300.147,415.999,176.996,22.222,153.377
C01509=1089.819,299.899,416.030,176.993,22.219,153.377
C01510=1089.814,299.651,416.060,176.990,22.216,153.377
C01511=1089.808,299.402,416.091,176.987,22.213,153.376
C01512=1089.802,299.155,416.122,176.984,22.210,153.376
C01513=1089.797,298.907,416.153,176.981,22.206,153.376
C01514=1089.791,298.659,416.183,176.978,22.203,153.375
C01515=1089.785,298.411,416.213,176.975,22.199,153.375
C01516=1089.780,298.163,416.244,176.972,22.196,153.375
C01517=1089.774,297.915,416.275,176.969,22.193,153.375
C01518=1089.769,297.667,416.305,176.966,22.190,153.374
C01519=1089.763,297.419,416.335,176.963,22.187,153.374
C01520=1089.758,297.171,416.366,176.960,22.183,153.374
C01521=1089.752,296.922,416.396,176.957,22.181,153.374
C01522=1089.746,296.674,416.427,176.954,22.177,153.373
C01523=1089.740,296.426,416.457,176.951,22.174,153.373
C01524=1089.734,296.179,416.487,176.948,22.171,153.373
C01525=1089.729,295.930,416.517,176.945,22.168,153.372
C01526=1089.723,295.682,416.547,176.942,22.165,153.372
C01527=1089.717,295.434,416.578,176.939,22.162,153.372
C01528=1089.712,295.186,416.609,176.936,22.159,153.372
C01529=1089.706,294.938,416.638,176.933,22.156,153.372
C01530=1089.701,294.690,416.669,176.930,22.153,153.371
C01531=1089.695,294.442,416.699,176.927,22.149,153.371
C01532=1089.689,294.194,416.729,176.924,22.146,153.371
C01533=1089.683,293.946,416.759,176.921,22.143,153.370
C01534=1089.678,293.698,416.789,176.918,22.140,153.370
C01535=1089.672,293.450,416.819,176.915,22.137,153.370
C01536=1089.666,293.202,416.849,176.912,22.134,153.370
C01537=1089.660,292.953,416.880,176.909,22.131,153.370
C01538=1089.654,292.705,416.910,176.906,22.128,153.369
C01539=1089.649,292.458,416.940,176.903,22.125,153.369
C01540=1089.643,292.209,416.970,176.900,22.122,153.369
C01541=1089.637,291.961,417.000,176.897,22.118,153.368
C01542=1089.631,291.713,417.030,176.894,22.115,153.368
C01543=1089.626,291.465,417.060,176.891,22.112,153.368
C01544=1089.620,291.217,417.090,176.888,22.109,153.368
C01545=1089.615,290.969,417.120,176.885,22.106,153.368
C01546=1089.610,290.721,417.149,176.882,22.103,153.367
C01547=1089.604,290.473,417.180,176.879,22.100,153.367
C01548=1089.594,290.090,417.226,176.875,22.095,153.367
C01549=1089.586,289.708,417.271,176.870,22.091,153.366
C01550=1089.577,289.326,417.317,176.865,22.086,153.366
C01551=1089.568,288.944,417.364,176.861,22.082,153.366
C01552=1089.563,288.695,417.393,176.858,22.078,153.365
C01553=1089.556,288.448,417.423,176.855,22.076,153.365
C01554=1089.551,288.199,417.453,176.852,22.073,153.365
C01555=1089.545,287.951,417.482,176.849,22.070,153.365
C01556=1089.540,287.702,417.512,176.846,22.067,153.365
C01557=1089.534,287.455,417.542,176.843,22.063,153.364
C01558=1089.528,287.206,417.571,176.840,22.061,153.364
C01559=1089.522,286.958,417.601,176.837,22.058,153.364
C01560=1089.516,286.710,417.631,176.834,22.055,153.364
C01561=1089.511,286.462,417.661,176.831,22.052,153.363
C01562=1089.505,286.214,417.690,176.828,22.048,153.363
C01563=1089.500,285.966,417.719,176.825,22.046,153.363
C01564=1089.494,285.717,417.749,176.822,22.043,153.363
C01565=1089.488,285.469,417.778,176.819,22.040,153.363
C01566=1089.482,285.221,417.808,176.816,22.037,153.362
C01567=1089.477,284.973,417.838,176.813,22.034,153.362
C01568=1089.471,284.725,417.867,176.810,22.031,153.362
C01569=1089.465,284.477,417.896,176.807,22.028,153.362
C01570=1089.460,284.229,417.926,176.804,22.025,153.361
C01571=1089.454,283.980,417.955,176.801,22.022,153.361
C01572=1089.448,283.732,417.984,176.798,22.019,153.361
C01573=1089.443,283.484,418.014,176.795,22.016,153.361
C01574=1089.437,283.235,418.044,176.792,22.013,153.361
C01575=1089.432,282.988,418.072,176.789,22.010,153.360
C01576=1089.426,282.739,418.102,176.787,22.008,153.360
C01577=1089.421,282.491,418.132,176.784,22.005,153.360
C01578=1089.414,282.243,418.161,176.781,22.001,153.360
C01579=1089.409,281.995,418.190,176.778,21.999,153.360
C01580=1089.404,281.747,418.220,176.775,21.996,153.359
C01581=1089.398,281.498,418.249,176.772,21.992,153.359
C01582=1089.392,281.250,418.278,176.769,21.990,153.359
C01583=1089.386,281.003,418.307,176.766,21.987,153.359
C01584=1089.381,280.754,418.337,176.763,21.984,153.358
C01585=1089.375,280.506,418.366,176.760,21.981,153.358
C01586=1089.369,280.258,418.395,176.757,21.978,153.358
C01587=1089.363,280.009,418.424,176.754,21.976,153.358
C01588=1089.358,279.761,418.453,176.751,21.972,153.358
C01589=1089.352,279.513,418.482,176.748,21.969,153.358
C01590=1089.347,279.265,418.512,176.745,21.967,153.357
C01591=1089.340,279.016,418.541,176.742,21.964,153.357
C01592=1089.335,278.769,418.570,176.739,21.960,153.357
C01593=1089.329,278.520,418.598,176.736,21.958,153.357
C01594=1089.324,278.271,418.628,176.733,21.955,153.357
C01595=1089.318,278.023,418.657,176.731,21.952,153.356
C01596=1089.313,277.775,418.685,176.728,21.949,153.356
C01597=1089.307,277.527,418.714,176.725,21.946,153.356
C01598=1089.301,277.279,418.743,176.722,21.944,153.356
C01599=1089.296,277.031,418.773,176.718,21.941,153.356
C01600=1089.287,276.657,418.816,176.714,21.936,153.355
C01601=1089.278,276.285,418.859,176.709,21.932,153.355
C01602=1089.270,275.912,418.903,176.706,21.928,153.355
C01603=1089.262,275.539,418.946,176.701,21.924,153.355
C01604=1089.256,275.291,418.975,176.698,21.920,153.354
C01605=1089.250,275.043,419.004,176.695,21.918,153.354
C01606=1089.245,274.794,419.033,176.692,21.915,153.354
C01607=1089.239,274.547,419.061,176.689,21.912,153.354
C01608=1089.233,274.298,419.090,176.687,21.910,153.354
C01609=1089.227,274.049,419.119,176.684,21.906,153.353
C01610=1089.222,273.801,419.147,176.681,21.904,153.353
C01611=1089.216,273.553,419.176,176.677,21.901,153.353
C01612=1089.210,273.305,419.204,176.674,21.898,153.353
C01613=1089.205,273.057,419.234,176.671,21.895,153.353
C01614=1089.199,272.808,419.262,176.669,21.893,153.352
C01615=1089.194,272.560,419.290,176.666,21.890,153.352
C01616=1089.187,272.312,419.319,176.663,21.887,153.352
C01617=1089.182,272.063,419.348,176.660,21.884,153.352
C01618=1089.177,271.815,419.377,176.657,21.881,153.352
C01619=1089.171,271.567,419.405,176.654,21.878,153.352
C01620=1089.165,271.319,419.433,176.651,21.875,153.351
C01621=1089.159,271.070,419.462,176.648,21.873,153.351
C01622=1089.154,270.822,419.490,176.645,21.870,153.351
C01623=1089.148,270.573,419.519,176.642,21.867,153.351
C01624=1089.142,270.325,419.548,176.639,21.864,153.351
C01625=1089.137,270.077,419.576,176.636,21.862,153.351
C01626=1089.131,269.828,419.604,176.634,21.859,153.350
C01627=1089.126,269.580,419.632,176.631,21.856,153.350
C01628=1089.119,269.332,419.661,176.628,21.854,153.350
C01629=1089.114,269.084,419.689,176.625,21.850,153.350
C01630=1089.108,268.835,419.718,176.622,21.847,153.350
C01631=1089.103,268.587,419.745,176.619,21.845,153.349
C01632=1089.096,268.339,419.775,176.616,21.842,153.349
C01633=1089.091,268.090,419.803,176.613,21.839,153.349
C01634=1089.086,267.842,419.831,176.610,21.837,153.349
C01635=1089.080,267.593,419.860,176.607,21.834,153.349
C01636=1089.075,267.345,419.888,176.604,21.831,153.349
C01637=1089.069,267.097,419.916,176.602,21.829,153.348
C01638=1089.063,266.849,419.944,176.599,21.826,153.348
C01639=1089.057,266.600,419.972,176.596,21.823,153.348
C01640=1089.052,266.352,420.001,176.592,21.820,153.348
C01641=1089.046,266.104,420.029,176.589,21.817,153.348
C01642=1089.041,265.856,420.057,176.587,21.815,153.348
C01643=1089.035,265.608,420.085,176.584,21.812,153.348
C01644=1089.029,265.359,420.114,176.581,21.809,153.347
C01645=1089.024,265.111,420.141,176.578,21.806,153.347
C01646=1089.018,264.862,420.170,176.575,21.803,153.347
C01647=1089.013,264.614,420.198,176.573,21.801,153.347
C01648=1089.007,264.365,420.226,176.569,21.798,153.347
C01649=1089.001,264.117,420.253,176.566,21.795,153.347
C01650=1088.995,263.868,420.281,176.563,21.793,153.346
C01651=1088.990,263.620,420.309,176.561,21.790,153.346
C01652=1088.980,263.250,420.351,176.556,21.786,153.346
C01653=1088.972,262.880,420.393,176.552,21.782,153.346
C01654=1088.963,262.511,420.434,176.548,21.778,153.346
C01655=1088.955,262.140,420.475,176.543,21.774,153.345
C01656=1088.949,261.892,420.503,176.540,21.771,153.345
C01657=1088.943,261.643,420.531,176.538,21.769,153.345
C01658=1088.938,261.395,420.559,176.535,21.767,153.345
C01659=1088.932,261.146,420.586,176.532,21.764,153.345
C01660=1088.926,260.898,420.614,176.528,21.761,153.345
C01661=1088.920,260.650,420.642,176.525,21.758,153.345
C01662=1088.914,260.402,420.670,176.523,21.756,153.344
C01663=1088.908,260.153,420.698,176.520,21.753,153.344
C01664=1088.903,259.904,420.725,176.517,21.750,153.344
C01665=1088.897,259.657,420.753,176.514,21.748,153.344
C01666=1088.891,259.408,420.781,176.511,21.745,153.344
C01667=1088.886,259.159,420.808,176.508,21.743,153.344
C01668=1088.880,258.912,420.836,176.505,21.740,153.344
C01669=1088.874,258.663,420.864,176.502,21.737,153.343
C01670=1088.869,258.414,420.891,176.500,21.734,153.343
C01671=1088.862,258.166,420.919,176.497,21.732,153.343
C01672=1088.857,257.917,420.946,176.494,21.729,153.343
C01673=1088.852,257.669,420.974,176.491,21.726,153.343
C01674=1088.845,257.420,421.002,176.488,21.724,153.343
C01675=1088.840,257.172,421.029,176.485,21.721,153.343
C01676=1088.834,256.924,421.057,176.482,21.718,153.342
C01677=1088.829,256.675,421.084,176.480,21.716,153.342
C01678=1088.823,256.427,421.112,176.477,21.713,153.342
C01679=1088.817,256.178,421.139,176.474,21.710,153.342
C01680=1088.812,255.930,421.167,176.471,21.708,153.342
C01681=1088.806,255.681,421.194,176.468,21.706,153.342
C01682=1088.800,255.433,421.222,176.465,21.703,153.342
C01683=1088.795,255.184,421.249,176.462,21.700,153.341
C01684=1088.789,254.937,421.276,176.459,21.697,153.341
C01685=1088.784,254.687,421.304,176.457,21.695,153.341
C01686=1088.778,254.440,421.331,176.454,21.692,153.341
C01687=1088.773,254.191,421.359,176.451,21.689,153.341
C01688=1088.767,253.943,421.385,176.448,21.687,153.341
C01689=1088.761,253.694,421.413,176.445,21.684,153.341
C01690=1088.755,253.445,421.440,176.442,21.681,153.341
C01691=1088.750,253.197,421.467,176.439,21.679,153.340
C01692=1088.744,252.949,421.495,176.437,21.676,153.340
C01693=1088.739,252.700,421.522,176.434,21.673,153.340
C01694=1088.733,252.451,421.550,176.431,21.671,153.340
C01695=1088.727,252.203,421.577,176.428,21.668,153.340
C01696=1088.722,251.955,421.604,176.425,21.665,153.340
C01697=1088.716,251.706,421.631,176.422,21.663,153.339
C01698=1088.711,251.458,421.659,176.419,21.660,153.339
C01699=1088.705,251.210,421.685,176.417,21.658,153.339
C01700=1088.700,250.960,421.713,176.414,21.655,153.339
C01701=1088.694,250.712,421.740,176.411,21.652,153.339
C01702=1088.689,250.463,421.767,176.408,21.650,153.339
C01703=1088.683,250.216,421.794,176.405,21.647,153.339
C01704=1088.675,249.843,421.835,176.401,21.643,153.338
C01705=1088.666,249.470,421.875,176.397,21.639,153.338
C01706=1088.657,249.097,421.916,176.392,21.635,153.338
C01707=1088.650,248.724,421.956,176.388,21.631,153.338
C01708=1088.644,248.476,421.983,176.385,21.628,153.338
C01709=1088.639,248.227,422.010,176.382,21.626,153.337
C01710=1088.633,247.979,422.037,176.380,21.623,153.337
C01711=1088.628,247.730,422.064,176.377,21.620,153.337
C01712=1088.622,247.481,422.091,176.374,21.617,153.337
C01713=1088.617,247.233,422.117,176.372,21.615,153.337
C01714=1088.611,246.984,422.145,176.369,21.612,153.337
C01715=1088.605,246.735,422.172,176.365,21.609,153.337
C01716=1088.599,246.487,422.198,176.363,21.607,153.336
C01717=1088.594,246.238,422.226,176.360,21.605,153.336
C01718=1088.589,245.990,422.252,176.357,21.602,153.336
C01719=1088.583,245.742,422.279,176.355,21.599,153.336
C01720=1088.577,245.493,422.306,176.352,21.597,153.336
C01721=1088.571,245.245,422.332,176.348,21.594,153.336
C01722=1088.566,244.996,422.359,176.346,21.592,153.336
C01723=1088.560,244.748,422.386,176.343,21.589,153.336
C01724=1088.555,244.500,422.413,176.340,21.586,153.335
C01725=1088.549,244.251,422.439,176.338,21.584,153.335
C01726=1088.544,244.002,422.467,176.335,21.581,153.335
C01727=1088.538,243.754,422.493,176.331,21.579,153.335
C01728=1088.533,243.505,422.519,176.329,21.576,153.335
C01729=1088.527,243.257,422.546,176.326,21.573,153.335
C01730=1088.521,243.008,422.572,176.324,21.571,153.335
C01731=1088.515,242.760,422.599,176.321,21.569,153.335
C01732=1088.510,242.511,422.625,176.318,21.566,153.334
C01733=1088.505,242.262,422.652,176.315,21.563,153.334
C01734=1088.499,242.014,422.679,176.312,21.560,153.334
C01735=1088.493,241.765,422.706,176.309,21.558,153.334
C01736=1088.487,241.516,422.732,176.307,21.556,153.334
C01737=1088.481,241.268,422.759,176.304,21.553,153.334
C01738=1088.476,241.019,422.785,176.301,21.550,153.334
C01739=1088.470,240.771,422.812,176.298,21.548,153.334
C01740=1088.464,240.522,422.838,176.295,21.545,153.333
C01741=1088.459,240.274,422.864,176.293,21.543,153.333
C01742=1088.453,240.026,422.891,176.290,21.540,153.333
C01743=1088.448,239.777,422.917,176.287,21.538,153.333
C01744=1088.442,239.529,422.943,176.284,21.535,153.333
C01745=1088.437,239.280,422.969,176.281,21.532,153.333
C01746=1088.431,239.031,422.996,176.278,21.530,153.333
C01747=1088.425,238.783,423.023,176.276,21.528,153.333
C01748=1088.420,238.534,423.048,176.273,21.525,153.332
C01749=1088.413,238.286,423.075,176.270,21.523,153.332
C01750=1088.408,238.037,423.100,176.267,21.520,153.332
C01751=1088.402,237.789,423.127,176.264,21.517,153.332
C01752=1088.396,237.540,423.153,176.262,21.515,153.332
C01753=1088.391,237.291,423.180,176.259,21.512,153.332
C01754=1088.385,237.042,423.206,176.257,21.510,153.332
C01755=1088.379,236.794,423.232,176.254,21.507,153.332
C01756=1088.371,236.414,423.272,176.249,21.503,153.332
C01757=1088.363,236.034,423.312,176.245,21.500,153.331
C01758=1088.354,235.655,423.352,176.240,21.495,153.331
C01759=1088.345,235.275,423.391,176.236,21.492,153.331
C01760=1088.340,235.026,423.418,176.233,21.489,153.331
C01761=1088.334,234.777,423.444,176.231,21.487,153.331
C01762=1088.329,234.529,423.469,176.228,21.484,153.330
C01763=1088.323,234.281,423.496,176.226,21.482,153.330
C01764=1088.318,234.032,423.522,176.223,21.479,153.330
C01765=1088.312,233.783,423.547,176.220,21.476,153.330
C01766=1088.306,233.535,423.574,176.217,21.474,153.330
C01767=1088.301,233.286,423.600,176.214,21.471,153.330
C01768=1088.296,233.037,423.625,176.212,21.469,153.330
C01769=1088.289,232.789,423.652,176.209,21.466,153.330
C01770=1088.284,232.540,423.677,176.206,21.464,153.330
C01771=1088.278,232.291,423.703,176.203,21.461,153.329
C01772=1088.273,232.042,423.729,176.200,21.459,153.329
C01773=1088.267,231.795,423.755,176.198,21.456,153.329
C01774=1088.261,231.546,423.781,176.195,21.454,153.329
C01775=1088.256,231.297,423.807,176.193,21.451,153.329
C01776=1088.250,231.048,423.833,176.190,21.449,153.329
C01777=1088.244,230.799,423.858,176.186,21.446,153.329
C01778=1088.239,230.551,423.884,176.184,21.444,153.329
C01779=1088.234,230.303,423.910,176.181,21.441,153.329
C01780=1088.227,230.054,423.936,176.179,21.439,153.328
C01781=1088.222,229.805,423.962,176.176,21.436,153.328
C01782=1088.216,229.557,423.987,176.173,21.434,153.328
C01783=1088.211,229.308,424.013,176.170,21.431,153.328
C01784=1088.205,229.059,424.038,176.168,21.429,153.328
C01785=1088.199,228.811,424.064,176.165,21.426,153.328
C01786=1088.194,228.562,424.090,176.162,21.424,153.328
C01787=1088.188,228.314,424.115,176.159,21.421,153.328
C01788=1088.183,228.065,424.141,176.156,21.419,153.328
C01789=1088.176,227.816,424.166,176.154,21.417,153.328
C01790=1088.171,227.567,424.192,176.151,21.414,153.327
C01791=1088.165,227.319,424.217,176.149,21.411,153.327
C01792=1088.160,227.070,424.243,176.145,21.409,153.327
C01793=1088.154,226.821,424.268,176.143,21.407,153.327
C01794=1088.149,226.573,424.294,176.140,21.404,153.327
C01795=1088.143,226.324,424.319,176.138,21.402,153.327
C01796=1088.137,226.075,424.345,176.135,21.399,153.327
C01797=1088.132,225.828,424.370,176.132,21.397,153.327
C01798=1088.126,225.579,424.396,176.129,21.394,153.327
C01799=1088.120,225.330,424.421,176.126,21.391,153.326
C01800=1088.114,225.081,424.447,176.124,21.389,153.326
C01801=1088.109,224.833,424.472,176.121,21.387,153.326
C01802=1088.104,224.583,424.497,176.119,21.384,153.326
C01803=1088.098,224.335,424.522,176.115,21.381,153.326
C01804=1088.093,224.086,424.548,176.113,21.379,153.326
C01805=1088.086,223.838,424.574,176.110,21.377,153.326
C01806=1088.081,223.589,424.599,176.108,21.374,153.326
C01807=1088.076,223.340,424.624,176.105,21.372,153.326
C01808=1088.067,222.952,424.664,176.101,21.368,153.325
C01809=1088.058,222.564,424.703,176.096,21.364,153.325
